LIN {X 0,Y 573.23,Z 214.707,A -85,B 0,C 180,E1 -2343.515,E2 -2343.515} C_VEL
LIN {X 0,Y 573.292,Z 214.696,A -85,B 0,C 180,E1 -2345.628,E2 -2345.628} C_VEL
LIN {X 0,Y 573.285,Z 214.699,A -85,B 0,C 180,E1 -2348.46,E2 -2348.46} C_VEL
LIN {X 0,Y 573.275,Z 214.705,A -85,B 0,C 180,E1 -2351.312,E2 -2351.312} C_VEL
LIN {X 0,Y 573.259,Z 214.704,A -85,B 0,C 180,E1 -2354.414,E2 -2354.414} C_VEL
LIN {X 0,Y 573.261,Z 214.7,A -85,B 0,C 180,E1 -2357.112,E2 -2357.112} C_VEL
LIN {X 0,Y 573.238,Z 214.703,A -85,B 0,C 180,E1 -2360.077,E2 -2360.077} C_VEL
LIN {X 0,Y 573.221,Z 214.707,A -85,B 0,C 180,E1 -2362.339,E2 -2362.339} C_VEL
LIN {X 0,Y 573.248,Z 214.702,A -85,B 0,C 180,E1 -2364.39,E2 -2364.39} C_VEL
LIN {X 0,Y 572.625,Z 214.783,A -85,B 0,C 180,E1 -2364.976,E2 -2364.976} C_VEL
LIN {X 0,Y 569.778,Z 215.141,A -85,B 0,C 180,E1 -2365.927,E2 -2365.927} C_VEL
LIN {X 0,Y 567.338,Z 215.445,A -85,B 0,C 180,E1 -2366.693,E2 -2366.693} C_VEL
LIN {X 0,Y 566.279,Z 215.573,A -85,B 0,C 180,E1 -2367.284,E2 -2367.284} C_VEL
LIN {X 0,Y 566.188,Z 215.583,A -85,B 0,C 180,E1 -2367.484,E2 -2367.484} C_VEL
LIN {X 0,Y 566.196,Z 215.58,A -85,B 0,C 180,E1 -2369.769,E2 -2369.769} C_VEL
LIN {X 0,Y 566.205,Z 215.585,A -85,B 0,C 180,E1 -2372.43,E2 -2372.43} C_VEL
LIN {X 0,Y 566.182,Z 215.582,A -85,B 0,C 180,E1 -2374.989,E2 -2374.989} C_VEL
LIN {X 0,Y 566.198,Z 215.584,A -85,B 0,C 180,E1 -2377.461,E2 -2377.461} C_VEL
LIN {X 0,Y 566.208,Z 215.581,A -85,B 0,C 180,E1 -2380.199,E2 -2380.199} C_VEL
LIN {X 0,Y 566.198,Z 215.58,A -85,B 0,C 180,E1 -2383.055,E2 -2383.055} C_VEL
LIN {X 0,Y 566.196,Z 215.581,A -85,B 0,C 180,E1 -2386.049,E2 -2386.049} C_VEL
LIN {X 0,Y 566.206,Z 215.58,A -85,B 0,C 180,E1 -2389.215,E2 -2389.215} C_VEL
LIN {X 0,Y 566.158,Z 215.588,A -85,B 0,C 180,E1 -2391.449,E2 -2391.449} C_VEL
LIN {X 0,Y 566.211,Z 219.363,A -85,B 0,C 180,E1 -2393.785,E2 -2393.785} C_VEL
LIN {X 0,Y 566.182,Z 223.459,A -85,B 0,C 180,E1 -2396.271,E2 -2396.271} C_VEL
LIN {X 0,Y 566.113,Z 227.943,A -85,B 0,C 180,E1 -2398.937,E2 -2398.937} C_VEL
LIN {X 0,Y 566.059,Z 232.969,A -85,B 0,C 180,E1 -2401.849,E2 -2401.849} C_VEL
LIN {X 0,Y 566.043,Z 238.59,A -85,B 0,C 180,E1 -2405.03,E2 -2405.03} C_VEL
LIN {X 0,Y 565.994,Z 242.827,A -85,B 0,C 180,E1 -2407.361,E2 -2407.361} C_VEL
LIN {X 0,Y 565.932,Z 247.064,A -85,B 0,C 180,E1 -2409.652,E2 -2409.652} C_VEL
LIN {X 0,Y 565.945,Z 251.369,A -85,B 0,C 180,E1 -2411.913,E2 -2411.913} C_VEL
LIN {X 0,Y 565.953,Z 256.885,A -85,B 0,C 180,E1 -2414.769,E2 -2414.769} C_VEL
LIN {X 0,Y 567.409,Z 265.07,A -85,B 0,C 180,E1 -2414.964,E2 -2414.964} C_VEL
LIN {X 0,Y 567.246,Z 279.422,A -85,B 0,C 180,E1 -2415.331,E2 -2415.331} C_VEL
LIN {X 0,Y 567.109,Z 293.099,A -85,B 0,C 180,E1 -2415.833,E2 -2415.833} C_VEL
LIN {X 0,Y 566.885,Z 306.271,A -85,B 0,C 180,E1 -2416.467,E2 -2416.467} C_VEL
LIN {X 0,Y 566.722,Z 318.211,A -85,B 0,C 180,E1 -2417.193,E2 -2417.193} C_VEL
LIN {X 0,Y 566.536,Z 330.289,A -85,B 0,C 180,E1 -2418.098,E2 -2418.098} C_VEL
LIN {X 0,Y 566.4,Z 341.502,A -85,B 0,C 180,E1 -2419.126,E2 -2419.126} C_VEL
LIN {X 0,Y 566.201,Z 350.968,A -85,B 0,C 180,E1 -2420.173,E2 -2420.173} C_VEL
LIN {X 0,Y 566.123,Z 359.1,A -85,B 0,C 180,E1 -2421.253,E2 -2421.253} C_VEL
LIN {X 0,Y 566.016,Z 366.883,A -85,B 0,C 180,E1 -2422.509,E2 -2422.509} C_VEL
LIN {X 0,Y 565.945,Z 372.324,A -85,B 0,C 180,E1 -2423.583,E2 -2423.583} C_VEL
LIN {X 0,Y 565.928,Z 376.8,A -85,B 0,C 180,E1 -2424.656,E2 -2424.656} C_VEL
LIN {X 0,Y 565.956,Z 380.312,A -85,B 0,C 180,E1 -2425.727,E2 -2425.727} C_VEL
LIN {X 0,Y 565.876,Z 383.744,A -85,B 0,C 180,E1 -2427.153,E2 -2427.153} C_VEL
LIN {X 0,Y 565.843,Z 385.785,A -85,B 0,C 180,E1 -2428.577,E2 -2428.577} C_VEL
LIN {X 0,Y 565.837,Z 386.496,A -85,B 0,C 180,E1 -2430,E2 -2430} C_VEL
LIN {X 0,Y 565.841,Z 385.88,A -85,B 0,C 180,E1 -2431.424,E2 -2431.424} C_VEL
LIN {X 0,Y 565.874,Z 383.922,A -85,B 0,C 180,E1 -2432.848,E2 -2432.848} C_VEL
LIN {X 0,Y 565.957,Z 380.576,A -85,B 0,C 180,E1 -2434.273,E2 -2434.273} C_VEL
LIN {X 0,Y 565.983,Z 375.747,A -85,B 0,C 180,E1 -2435.701,E2 -2435.701} C_VEL
LIN {X 0,Y 565.981,Z 369.281,A -85,B 0,C 180,E1 -2437.133,E2 -2437.133} C_VEL
LIN {X 0,Y 566.093,Z 362.081,A -85,B 0,C 180,E1 -2438.388,E2 -2438.388} C_VEL
LIN {X 0,Y 566.172,Z 354.54,A -85,B 0,C 180,E1 -2439.467,E2 -2439.467} C_VEL
LIN {X 0,Y 566.29,Z 345.484,A -85,B 0,C 180,E1 -2440.548,E2 -2440.548} C_VEL
LIN {X 0,Y 566.471,Z 334.519,A -85,B 0,C 180,E1 -2441.631,E2 -2441.631} C_VEL
LIN {X 0,Y 566.644,Z 323.343,A -85,B 0,C 180,E1 -2442.536,E2 -2442.536} C_VEL
LIN {X 0,Y 566.854,Z 310.99,A -85,B 0,C 180,E1 -2443.351,E2 -2443.351} C_VEL
LIN {X 0,Y 566.995,Z 299.106,A -85,B 0,C 180,E1 -2443.987,E2 -2443.987} C_VEL
LIN {X 0,Y 567.178,Z 285.584,A -85,B 0,C 180,E1 -2444.551,E2 -2444.551} C_VEL
LIN {X 0,Y 567.354,Z 272.078,A -85,B 0,C 180,E1 -2444.965,E2 -2444.965} C_VEL
LIN {X 0,Y 567.197,Z 263.074,A -85,B 0,C 180,E1 -2445.172,E2 -2445.172} C_VEL
LIN {X 0,Y 565.917,Z 256.881,A -85,B 0,C 180,E1 -2445.325,E2 -2445.325} C_VEL
LIN {X 0,Y 565.944,Z 251.541,A -85,B 0,C 180,E1 -2448.087,E2 -2448.087} C_VEL
LIN {X 0,Y 565.933,Z 247.234,A -85,B 0,C 180,E1 -2450.348,E2 -2450.348} C_VEL
LIN {X 0,Y 566.046,Z 241.879,A -85,B 0,C 180,E1 -2453.251,E2 -2453.251} C_VEL
LIN {X 0,Y 566.008,Z 237.377,A -85,B 0,C 180,E1 -2455.759,E2 -2455.759} C_VEL
LIN {X 0,Y 566.066,Z 233.084,A -85,B 0,C 180,E1 -2458.176,E2 -2458.176} C_VEL
LIN {X 0,Y 566.12,Z 227.472,A -85,B 0,C 180,E1 -2461.427,E2 -2461.427} C_VEL
LIN {X 0,Y 566.181,Z 223.231,A -85,B 0,C 180,E1 -2463.958,E2 -2463.958} C_VEL
LIN {X 0,Y 566.226,Z 218.933,A -85,B 0,C 180,E1 -2466.568,E2 -2466.568} C_VEL
LIN {X 0,Y 566.148,Z 215.738,A -85,B 0,C 180,E1 -2468.55,E2 -2468.55} C_VEL
LIN {X 0,Y 566.206,Z 215.581,A -85,B 0,C 180,E1 -2470.785,E2 -2470.785} C_VEL
LIN {X 0,Y 566.197,Z 215.58,A -85,B 0,C 180,E1 -2473.951,E2 -2473.951} C_VEL
LIN {X 0,Y 566.204,Z 215.58,A -85,B 0,C 180,E1 -2477.083,E2 -2477.083} C_VEL
LIN {X 0,Y 566.212,Z 215.578,A -85,B 0,C 180,E1 -2480.315,E2 -2480.315} C_VEL
LIN {X 0,Y 566.203,Z 215.579,A -85,B 0,C 180,E1 -2483.43,E2 -2483.43} C_VEL
LIN {X 0,Y 566.201,Z 215.583,A -85,B 0,C 180,E1 -2486.268,E2 -2486.268} C_VEL
LIN {X 0,Y 566.183,Z 215.584,A -85,B 0,C 180,E1 -2488.926,E2 -2488.926} C_VEL
LIN {X 0,Y 566.197,Z 215.58,A -85,B 0,C 180,E1 -2491.856,E2 -2491.856} C_VEL
LIN {X 0,Y 566.217,Z 215.582,A -85,B 0,C 180,E1 -2494.251,E2 -2494.251} C_VEL
LIN {X 0,Y 566.171,Z 215.583,A -85,B 0,C 180,E1 -2496.72,E2 -2496.72} C_VEL
LIN {X 0,Y 566.205,Z 215.579,A -85,B 0,C 180,E1 -2499.662,E2 -2499.662} C_VEL
LIN {X 0,Y 566.201,Z 215.581,A -85,B 0,C 180,E1 -2502.668,E2 -2502.668} C_VEL
LIN {X 0,Y 566.231,Z 215.58,A -85,B 0,C 180,E1 -2505.627,E2 -2505.627} C_VEL
LIN {X 0,Y 566.239,Z 215.581,A -85,B 0,C 180,E1 -2508.676,E2 -2508.676} C_VEL
LIN {X 0,Y 566.208,Z 215.579,A -85,B 0,C 180,E1 -2511.434,E2 -2511.434} C_VEL
LIN {X 0,Y 566.261,Z 215.572,A -85,B 0,C 180,E1 -2514.302,E2 -2514.302} C_VEL
LIN {X 0,Y 566.264,Z 215.572,A -85,B 0,C 180,E1 -2517.866,E2 -2517.866} C_VEL
LIN {X 0,Y 566.303,Z 215.567,A -85,B 0,C 180,E1 -2520.711,E2 -2520.711} C_VEL
LIN {X 0,Y 566.276,Z 215.571,A -85,B 0,C 180,E1 -2522.845,E2 -2522.845} C_VEL
LIN {X 0,Y 566.245,Z 215.574,A -85,B 0,C 180,E1 -2525.698,E2 -2525.698} C_VEL
LIN {X 0,Y 566.195,Z 215.582,A -85,B 0,C 180,E1 -2528.566,E2 -2528.566} C_VEL
LIN {X 0,Y 566.246,Z 215.58,A -85,B 0,C 180,E1 -2531.454,E2 -2531.454} C_VEL
LIN {X 0,Y 566.241,Z 215.579,A -85,B 0,C 180,E1 -2534.507,E2 -2534.507} C_VEL
LIN {X 0,Y 566.174,Z 215.583,A -85,B 0,C 180,E1 -2537.332,E2 -2537.332} C_VEL
LIN {X 0,Y 566.205,Z 215.585,A -85,B 0,C 180,E1 -2539.581,E2 -2539.581} C_VEL
LIN {X 0,Y 566.198,Z 215.58,A -85,B 0,C 180,E1 -2541.862,E2 -2541.862} C_VEL
LIN {X 0,Y 566.222,Z 215.576,A -85,B 0,C 180,E1 -2545.03,E2 -2545.03} C_VEL
LIN {X 0,Y 566.162,Z 215.587,A -85,B 0,C 180,E1 -2547.342,E2 -2547.342} C_VEL
LIN {X 0,Y 566.175,Z 215.583,A -85,B 0,C 180,E1 -2549.77,E2 -2549.77} C_VEL
LIN {X 0,Y 566.212,Z 215.584,A -85,B 0,C 180,E1 -2552.431,E2 -2552.431} C_VEL
LIN {X 0,Y 566.172,Z 215.584,A -85,B 0,C 180,E1 -2554.988,E2 -2554.988} C_VEL
LIN {X 0,Y 566.192,Z 215.586,A -85,B 0,C 180,E1 -2557.461,E2 -2557.461} C_VEL
LIN {X 0,Y 566.209,Z 215.581,A -85,B 0,C 180,E1 -2560.199,E2 -2560.199} C_VEL
LIN {X 0,Y 566.203,Z 215.581,A -85,B 0,C 180,E1 -2563.054,E2 -2563.054} C_VEL
LIN {X 0,Y 566.157,Z 215.586,A -85,B 0,C 180,E1 -2566.053,E2 -2566.053} C_VEL
LIN {X 0,Y 566.168,Z 215.589,A -85,B 0,C 180,E1 -2568.86,E2 -2568.86} C_VEL
LIN {X 0,Y 566.24,Z 215.762,A -85,B 0,C 180,E1 -2570.728,E2 -2570.728} C_VEL
LIN {X 0,Y 566.486,Z 219.701,A -85,B 0,C 180,E1 -2572.561,E2 -2572.561} C_VEL
LIN {X 0,Y 566.391,Z 226.653,A -85,B 0,C 180,E1 -2575.626,E2 -2575.626} C_VEL
LIN {X 0,Y 566.34,Z 233.716,A -85,B 0,C 180,E1 -2578.587,E2 -2578.587} C_VEL
LIN {X 0,Y 566.215,Z 239.77,A -85,B 0,C 180,E1 -2581.048,E2 -2581.048} C_VEL
LIN {X 0,Y 566.161,Z 246.859,A -85,B 0,C 180,E1 -2583.853,E2 -2583.853} C_VEL
LIN {X 0,Y 566.078,Z 253.937,A -85,B 0,C 180,E1 -2586.591,E2 -2586.591} C_VEL
LIN {X 0,Y 566.043,Z 261.995,A -85,B 0,C 180,E1 -2589.656,E2 -2589.656} C_VEL
LIN {X 0,Y 565.975,Z 269.986,A -85,B 0,C 180,E1 -2592.661,E2 -2592.661} C_VEL
LIN {X 0,Y 565.935,Z 275.545,A -85,B 0,C 180,E1 -2594.713,E2 -2594.713} C_VEL
LIN {X 0,Y 567.413,Z 283.017,A -85,B 0,C 180,E1 -2594.877,E2 -2594.877} C_VEL
LIN {X 0,Y 567.263,Z 297.785,A -85,B 0,C 180,E1 -2595.237,E2 -2595.237} C_VEL
LIN {X 0,Y 567.045,Z 311.961,A -85,B 0,C 180,E1 -2595.739,E2 -2595.739} C_VEL
LIN {X 0,Y 566.872,Z 325.392,A -85,B 0,C 180,E1 -2596.375,E2 -2596.375} C_VEL
LIN {X 0,Y 566.721,Z 337.512,A -85,B 0,C 180,E1 -2597.102,E2 -2597.102} C_VEL
LIN {X 0,Y 566.542,Z 349.749,A -85,B 0,C 180,E1 -2598.007,E2 -2598.007} C_VEL
LIN {X 0,Y 566.433,Z 360.501,A -85,B 0,C 180,E1 -2598.98,E2 -2598.98} C_VEL
LIN {X 0,Y 566.206,Z 369.851,A -85,B 0,C 180,E1 -2599.993,E2 -2599.993} C_VEL
LIN {X 0,Y 566.137,Z 378.172,A -85,B 0,C 180,E1 -2601.073,E2 -2601.073} C_VEL
LIN {X 0,Y 566.046,Z 386.127,A -85,B 0,C 180,E1 -2602.33,E2 -2602.33} C_VEL
LIN {X 0,Y 565.944,Z 392.527,A -85,B 0,C 180,E1 -2603.583,E2 -2603.583} C_VEL
LIN {X 0,Y 565.927,Z 396.961,A -85,B 0,C 180,E1 -2604.656,E2 -2604.656} C_VEL
LIN {X 0,Y 565.957,Z 400.443,A -85,B 0,C 180,E1 -2605.727,E2 -2605.727} C_VEL
LIN {X 0,Y 565.874,Z 403.832,A -85,B 0,C 180,E1 -2607.152,E2 -2607.152} C_VEL
LIN {X 0,Y 565.841,Z 405.833,A -85,B 0,C 180,E1 -2608.576,E2 -2608.576} C_VEL
LIN {X 0,Y 565.837,Z 406.5,A -85,B 0,C 180,E1 -2610,E2 -2610} C_VEL
LIN {X 0,Y 565.841,Z 405.834,A -85,B 0,C 180,E1 -2611.423,E2 -2611.423} C_VEL
LIN {X 0,Y 565.874,Z 403.834,A -85,B 0,C 180,E1 -2612.848,E2 -2612.848} C_VEL
LIN {X 0,Y 565.957,Z 400.445,A -85,B 0,C 180,E1 -2614.273,E2 -2614.273} C_VEL
LIN {X 0,Y 565.985,Z 395.568,A -85,B 0,C 180,E1 -2615.701,E2 -2615.701} C_VEL
LIN {X 0,Y 565.995,Z 391.044,A -85,B 0,C 180,E1 -2616.739,E2 -2616.739} C_VEL
LIN {X 0,Y 566.047,Z 384.037,A -85,B 0,C 180,E1 -2618.029,E2 -2618.029} C_VEL
LIN {X 0,Y 566.177,Z 375.558,A -85,B 0,C 180,E1 -2619.286,E2 -2619.286} C_VEL
LIN {X 0,Y 566.294,Z 366.707,A -85,B 0,C 180,E1 -2620.367,E2 -2620.367} C_VEL
LIN {X 0,Y 566.485,Z 355.989,A -85,B 0,C 180,E1 -2621.449,E2 -2621.449} C_VEL
LIN {X 0,Y 566.653,Z 345.14,A -85,B 0,C 180,E1 -2622.354,E2 -2622.354} C_VEL
LIN {X 0,Y 566.74,Z 333.256,A -85,B 0,C 180,E1 -2623.171,E2 -2623.171} C_VEL
LIN {X 0,Y 566.979,Z 320.096,A -85,B 0,C 180,E1 -2623.896,E2 -2623.896} C_VEL
LIN {X 0,Y 567.184,Z 307.303,A -85,B 0,C 180,E1 -2624.445,E2 -2624.445} C_VEL
LIN {X 0,Y 567.327,Z 293.409,A -85,B 0,C 180,E1 -2624.887,E2 -2624.887} C_VEL
LIN {X 0,Y 567.245,Z 282.071,A -85,B 0,C 180,E1 -2625.146,E2 -2625.146} C_VEL
LIN {X 0,Y 565.934,Z 275.48,A -85,B 0,C 180,E1 -2625.301,E2 -2625.301} C_VEL
LIN {X 0,Y 565.986,Z 267.989,A -85,B 0,C 180,E1 -2628.085,E2 -2628.085} C_VEL
LIN {X 0,Y 566.071,Z 259.998,A -85,B 0,C 180,E1 -2631.103,E2 -2631.103} C_VEL
LIN {X 0,Y 566.111,Z 251.897,A -85,B 0,C 180,E1 -2634.185,E2 -2634.185} C_VEL
LIN {X 0,Y 566.21,Z 243.8,A -85,B 0,C 180,E1 -2637.339,E2 -2637.339} C_VEL
LIN {X 0,Y 566.294,Z 235.712,A -85,B 0,C 180,E1 -2640.586,E2 -2640.586} C_VEL
LIN {X 0,Y 566.355,Z 229.675,A -85,B 0,C 180,E1 -2643.093,E2 -2643.093} C_VEL
LIN {X 0,Y 566.391,Z 223.657,A -85,B 0,C 180,E1 -2645.676,E2 -2645.676} C_VEL
LIN {X 0,Y 566.444,Z 217.719,A -85,B 0,C 180,E1 -2648.343,E2 -2648.343} C_VEL
LIN {X 0,Y 566.219,Z 215.582,A -85,B 0,C 180,E1 -2649.377,E2 -2649.377} C_VEL
LIN {X 0,Y 566.173,Z 215.584,A -85,B 0,C 180,E1 -2652.091,E2 -2652.091} C_VEL
LIN {X 0,Y 566.165,Z 215.587,A -85,B 0,C 180,E1 -2655.037,E2 -2655.037} C_VEL
LIN {X 0,Y 566.212,Z 215.584,A -85,B 0,C 180,E1 -2657.913,E2 -2657.913} C_VEL
LIN {X 0,Y 566.214,Z 215.581,A -85,B 0,C 180,E1 -2660.726,E2 -2660.726} C_VEL
LIN {X 0,Y 566.18,Z 215.583,A -85,B 0,C 180,E1 -2663.429,E2 -2663.429} C_VEL
LIN {X 0,Y 566.213,Z 215.581,A -85,B 0,C 180,E1 -2666.266,E2 -2666.266} C_VEL
LIN {X 0,Y 566.196,Z 215.584,A -85,B 0,C 180,E1 -2668.923,E2 -2668.923} C_VEL
LIN {X 0,Y 566.171,Z 215.584,A -85,B 0,C 180,E1 -2671.855,E2 -2671.855} C_VEL
LIN {X 0,Y 566.239,Z 215.575,A -85,B 0,C 180,E1 -2675.039,E2 -2675.039} C_VEL
LIN {X 0,Y 566.196,Z 215.58,A -85,B 0,C 180,E1 -2678.138,E2 -2678.138} C_VEL
LIN {X 0,Y 566.233,Z 215.581,A -85,B 0,C 180,E1 -2680.614,E2 -2680.614} C_VEL
LIN {X 0,Y 566.167,Z 215.585,A -85,B 0,C 180,E1 -2683.411,E2 -2683.411} C_VEL
LIN {X 0,Y 566.24,Z 215.578,A -85,B 0,C 180,E1 -2685.627,E2 -2685.627} C_VEL
LIN {X 0,Y 566.238,Z 215.58,A -85,B 0,C 180,E1 -2688.675,E2 -2688.675} C_VEL
LIN {X 0,Y 566.196,Z 215.581,A -85,B 0,C 180,E1 -2691.434,E2 -2691.434} C_VEL
LIN {X 0,Y 566.243,Z 215.574,A -85,B 0,C 180,E1 -2694.302,E2 -2694.302} C_VEL
LIN {X 0,Y 566.276,Z 215.572,A -85,B 0,C 180,E1 -2697.155,E2 -2697.155} C_VEL
LIN {X 0,Y 566.293,Z 215.575,A -85,B 0,C 180,E1 -2700,E2 -2700} C_VEL
LIN {X 0,Y 566.258,Z 215.574,A -85,B 0,C 180,E1 -2702.846,E2 -2702.846} C_VEL
LIN {X 0,Y 566.259,Z 215.572,A -85,B 0,C 180,E1 -2705.698,E2 -2705.698} C_VEL
LIN {X 0,Y 566.229,Z 215.577,A -85,B 0,C 180,E1 -2708.566,E2 -2708.566} C_VEL
LIN {X 0,Y 566.242,Z 215.579,A -85,B 0,C 180,E1 -2711.454,E2 -2711.454} C_VEL
LIN {X 0,Y 566.215,Z 215.583,A -85,B 0,C 180,E1 -2714.498,E2 -2714.498} C_VEL
LIN {X 0,Y 566.201,Z 215.58,A -85,B 0,C 180,E1 -2717.332,E2 -2717.332} C_VEL
LIN {X 0,Y 566.205,Z 215.579,A -85,B 0,C 180,E1 -2720.338,E2 -2720.338} C_VEL
LIN {X 0,Y 566.168,Z 215.584,A -85,B 0,C 180,E1 -2723.28,E2 -2723.28} C_VEL
LIN {X 0,Y 566.213,Z 215.582,A -85,B 0,C 180,E1 -2725.749,E2 -2725.749} C_VEL
LIN {X 0,Y 566.188,Z 215.583,A -85,B 0,C 180,E1 -2727.484,E2 -2727.484} C_VEL
LIN {X 0,Y 565.508,Z 215.667,A -85,B 0,C 180,E1 -2728.078,E2 -2728.078} C_VEL
LIN {X 0,Y 562.646,Z 216.027,A -85,B 0,C 180,E1 -2729.042,E2 -2729.042} C_VEL
LIN {X 0,Y 560.24,Z 216.324,A -85,B 0,C 180,E1 -2729.818,E2 -2729.818} C_VEL
LIN {X 0,Y 559.214,Z 216.452,A -85,B 0,C 180,E1 -2730.416,E2 -2730.416} C_VEL
LIN {X 0,Y 559.134,Z 216.46,A -85,B 0,C 180,E1 -2730.619,E2 -2730.619} C_VEL
LIN {X 0,Y 559.154,Z 216.46,A -85,B 0,C 180,E1 -2732.716,E2 -2732.716} C_VEL
LIN {X 0,Y 559.13,Z 216.463,A -85,B 0,C 180,E1 -2735.324,E2 -2735.324} C_VEL
LIN {X 0,Y 559.133,Z 216.46,A -85,B 0,C 180,E1 -2738.018,E2 -2738.018} C_VEL
LIN {X 0,Y 559.128,Z 216.464,A -85,B 0,C 180,E1 -2740.815,E2 -2740.815} C_VEL
LIN {X 0,Y 559.139,Z 216.466,A -85,B 0,C 180,E1 -2743.734,E2 -2743.734} C_VEL
LIN {X 0,Y 559.147,Z 216.462,A -85,B 0,C 180,E1 -2746.804,E2 -2746.804} C_VEL
LIN {X 0,Y 559.157,Z 216.458,A -85,B 0,C 180,E1 -2749.188,E2 -2749.188} C_VEL
LIN {X 0,Y 559.124,Z 216.463,A -85,B 0,C 180,E1 -2751.198,E2 -2751.198} C_VEL
LIN {X 0,Y 559.201,Z 218.824,A -85,B 0,C 180,E1 -2752.896,E2 -2752.896} C_VEL
LIN {X 0,Y 559.148,Z 223.949,A -85,B 0,C 180,E1 -2756.054,E2 -2756.054} C_VEL
LIN {X 0,Y 559.064,Z 228.806,A -85,B 0,C 180,E1 -2758.975,E2 -2758.975} C_VEL
LIN {X 0,Y 558.981,Z 233.38,A -85,B 0,C 180,E1 -2761.655,E2 -2761.655} C_VEL
LIN {X 0,Y 558.965,Z 238.679,A -85,B 0,C 180,E1 -2764.692,E2 -2764.692} C_VEL
LIN {X 0,Y 558.944,Z 242.914,A -85,B 0,C 180,E1 -2767.059,E2 -2767.059} C_VEL
LIN {X 0,Y 558.854,Z 247.126,A -85,B 0,C 180,E1 -2769.383,E2 -2769.383} C_VEL
LIN {X 0,Y 558.854,Z 251.37,A -85,B 0,C 180,E1 -2771.676,E2 -2771.676} C_VEL
LIN {X 0,Y 558.852,Z 256.887,A -85,B 0,C 180,E1 -2774.57,E2 -2774.57} C_VEL
LIN {X 0,Y 560.536,Z 265.968,A -85,B 0,C 180,E1 -2774.793,E2 -2774.793} C_VEL
LIN {X 0,Y 560.389,Z 279.941,A -85,B 0,C 180,E1 -2775.163,E2 -2775.163} C_VEL
LIN {X 0,Y 560.209,Z 294.189,A -85,B 0,C 180,E1 -2775.701,E2 -2775.701} C_VEL
LIN {X 0,Y 559.94,Z 307.872,A -85,B 0,C 180,E1 -2776.388,E2 -2776.388} C_VEL
LIN {X 0,Y 559.716,Z 320.802,A -85,B 0,C 180,E1 -2777.214,E2 -2777.214} C_VEL
LIN {X 0,Y 559.523,Z 332.432,A -85,B 0,C 180,E1 -2778.131,E2 -2778.131} C_VEL
LIN {X 0,Y 559.351,Z 342.956,A -85,B 0,C 180,E1 -2779.137,E2 -2779.137} C_VEL
LIN {X 0,Y 559.151,Z 352.457,A -85,B 0,C 180,E1 -2780.231,E2 -2780.231} C_VEL
LIN {X 0,Y 559.029,Z 361.525,A -85,B 0,C 180,E1 -2781.505,E2 -2781.505} C_VEL
LIN {X 0,Y 558.908,Z 368.829,A -85,B 0,C 180,E1 -2782.776,E2 -2782.776} C_VEL
LIN {X 0,Y 558.886,Z 373.939,A -85,B 0,C 180,E1 -2783.864,E2 -2783.864} C_VEL
LIN {X 0,Y 558.821,Z 379.25,A -85,B 0,C 180,E1 -2785.311,E2 -2785.311} C_VEL
LIN {X 0,Y 558.825,Z 382.209,A -85,B 0,C 180,E1 -2786.395,E2 -2786.395} C_VEL
LIN {X 0,Y 558.744,Z 384.935,A -85,B 0,C 180,E1 -2787.838,E2 -2787.838} C_VEL
LIN {X 0,Y 558.737,Z 386.306,A -85,B 0,C 180,E1 -2789.279,E2 -2789.279} C_VEL
LIN {X 0,Y 558.739,Z 386.354,A -85,B 0,C 180,E1 -2790.721,E2 -2790.721} C_VEL
LIN {X 0,Y 558.742,Z 385.07,A -85,B 0,C 180,E1 -2792.163,E2 -2792.163} C_VEL
LIN {X 0,Y 558.825,Z 382.426,A -85,B 0,C 180,E1 -2793.605,E2 -2793.605} C_VEL
LIN {X 0,Y 558.821,Z 379.513,A -85,B 0,C 180,E1 -2794.689,E2 -2794.689} C_VEL
LIN {X 0,Y 558.883,Z 374.321,A -85,B 0,C 180,E1 -2796.136,E2 -2796.136} C_VEL
LIN {X 0,Y 558.907,Z 369.278,A -85,B 0,C 180,E1 -2797.224,E2 -2797.224} C_VEL
LIN {X 0,Y 559.029,Z 362.078,A -85,B 0,C 180,E1 -2798.495,E2 -2798.495} C_VEL
LIN {X 0,Y 559.124,Z 354.537,A -85,B 0,C 180,E1 -2799.587,E2 -2799.587} C_VEL
LIN {X 0,Y 559.288,Z 345.478,A -85,B 0,C 180,E1 -2800.682,E2 -2800.682} C_VEL
LIN {X 0,Y 559.482,Z 334.512,A -85,B 0,C 180,E1 -2801.778,E2 -2801.778} C_VEL
LIN {X 0,Y 559.679,Z 323.336,A -85,B 0,C 180,E1 -2802.695,E2 -2802.695} C_VEL
LIN {X 0,Y 559.921,Z 310.983,A -85,B 0,C 180,E1 -2803.52,E2 -2803.52} C_VEL
LIN {X 0,Y 560.106,Z 299.096,A -85,B 0,C 180,E1 -2804.163,E2 -2804.163} C_VEL
LIN {X 0,Y 560.293,Z 286.039,A -85,B 0,C 180,E1 -2804.717,E2 -2804.717} C_VEL
LIN {X 0,Y 560.489,Z 272.334,A -85,B 0,C 180,E1 -2805.146,E2 -2805.146} C_VEL
LIN {X 0,Y 560.381,Z 264.367,A -85,B 0,C 180,E1 -2805.334,E2 -2805.334} C_VEL
LIN {X 0,Y 558.844,Z 256.88,A -85,B 0,C 180,E1 -2805.524,E2 -2805.524} C_VEL
LIN {X 0,Y 558.854,Z 251.54,A -85,B 0,C 180,E1 -2808.324,E2 -2808.324} C_VEL
LIN {X 0,Y 558.853,Z 247.29,A -85,B 0,C 180,E1 -2810.617,E2 -2810.617} C_VEL
LIN {X 0,Y 558.95,Z 242.295,A -85,B 0,C 180,E1 -2813.383,E2 -2813.383} C_VEL
LIN {X 0,Y 558.931,Z 237.446,A -85,B 0,C 180,E1 -2816.11,E2 -2816.11} C_VEL
LIN {X 0,Y 559.018,Z 233.198,A -85,B 0,C 180,E1 -2818.538,E2 -2818.538} C_VEL
LIN {X 0,Y 559.078,Z 228.558,A -85,B 0,C 180,E1 -2821.261,E2 -2821.261} C_VEL
LIN {X 0,Y 559.134,Z 223.286,A -85,B 0,C 180,E1 -2824.446,E2 -2824.446} C_VEL
LIN {X 0,Y 559.202,Z 218.976,A -85,B 0,C 180,E1 -2827.104,E2 -2827.104} C_VEL
LIN {X 0,Y 559.117,Z 216.466,A -85,B 0,C 180,E1 -2828.801,E2 -2828.801} C_VEL
LIN {X 0,Y 559.163,Z 216.46,A -85,B 0,C 180,E1 -2831.051,E2 -2831.051} C_VEL
LIN {X 0,Y 559.141,Z 216.46,A -85,B 0,C 180,E1 -2833.734,E2 -2833.734} C_VEL
LIN {X 0,Y 559.149,Z 216.46,A -85,B 0,C 180,E1 -2836.804,E2 -2836.804} C_VEL
LIN {X 0,Y 559.178,Z 216.455,A -85,B 0,C 180,E1 -2840.134,E2 -2840.134} C_VEL
LIN {X 0,Y 559.144,Z 216.464,A -85,B 0,C 180,E1 -2842.892,E2 -2842.892} C_VEL
LIN {X 0,Y 559.16,Z 216.463,A -85,B 0,C 180,E1 -2846.052,E2 -2846.052} C_VEL
LIN {X 0,Y 559.148,Z 216.461,A -85,B 0,C 180,E1 -2848.98,E2 -2848.98} C_VEL
LIN {X 0,Y 559.147,Z 216.458,A -85,B 0,C 180,E1 -2851.624,E2 -2851.624} C_VEL
LIN {X 0,Y 559.184,Z 216.457,A -85,B 0,C 180,E1 -2853.903,E2 -2853.903} C_VEL
LIN {X 0,Y 559.141,Z 216.459,A -85,B 0,C 180,E1 -2856.572,E2 -2856.572} C_VEL
LIN {X 0,Y 559.175,Z 216.456,A -85,B 0,C 180,E1 -2859.395,E2 -2859.395} C_VEL
LIN {X 0,Y 559.14,Z 216.46,A -85,B 0,C 180,E1 -2861.685,E2 -2861.685} C_VEL
LIN {X 0,Y 559.167,Z 216.461,A -85,B 0,C 180,E1 -2863.948,E2 -2863.948} C_VEL
LIN {X 0,Y 559.165,Z 216.456,A -85,B 0,C 180,E1 -2866.184,E2 -2866.184} C_VEL
LIN {X 0,Y 559.193,Z 216.454,A -85,B 0,C 180,E1 -2869.133,E2 -2869.133} C_VEL
LIN {X 0,Y 559.199,Z 216.457,A -85,B 0,C 180,E1 -2872.053,E2 -2872.053} C_VEL
LIN {X 0,Y 559.254,Z 216.448,A -85,B 0,C 180,E1 -2874.953,E2 -2874.953} C_VEL
LIN {X 0,Y 559.237,Z 216.447,A -85,B 0,C 180,E1 -2877.839,E2 -2877.839} C_VEL
LIN {X 0,Y 559.273,Z 216.443,A -85,B 0,C 180,E1 -2880.72,E2 -2880.72} C_VEL
LIN {X 0,Y 559.242,Z 216.447,A -85,B 0,C 180,E1 -2882.881,E2 -2882.881} C_VEL
LIN {X 0,Y 559.214,Z 216.45,A -85,B 0,C 180,E1 -2885.77,E2 -2885.77} C_VEL
LIN {X 0,Y 559.162,Z 216.457,A -85,B 0,C 180,E1 -2888.675,E2 -2888.675} C_VEL
LIN {X 0,Y 559.21,Z 216.454,A -85,B 0,C 180,E1 -2891.6,E2 -2891.6} C_VEL
LIN {X 0,Y 559.205,Z 216.457,A -85,B 0,C 180,E1 -2894.595,E2 -2894.595} C_VEL
LIN {X 0,Y 559.124,Z 216.463,A -85,B 0,C 180,E1 -2897.558,E2 -2897.558} C_VEL
LIN {X 0,Y 559.168,Z 216.458,A -85,B 0,C 180,E1 -2899.838,E2 -2899.838} C_VEL
LIN {X 0,Y 559.145,Z 216.459,A -85,B 0,C 180,E1 -2902.153,E2 -2902.153} C_VEL
LIN {X 0,Y 559.164,Z 216.455,A -85,B 0,C 180,E1 -2905.183,E2 -2905.183} C_VEL
LIN {X 0,Y 559.114,Z 216.462,A -85,B 0,C 180,E1 -2908.37,E2 -2908.37} C_VEL
LIN {X 0,Y 559.153,Z 216.459,A -85,B 0,C 180,E1 -2911.274,E2 -2911.274} C_VEL
LIN {X 0,Y 559.167,Z 216.46,A -85,B 0,C 180,E1 -2913.949,E2 -2913.949} C_VEL
LIN {X 0,Y 559.131,Z 216.465,A -85,B 0,C 180,E1 -2917.109,E2 -2917.109} C_VEL
LIN {X 0,Y 559.163,Z 216.457,A -85,B 0,C 180,E1 -2919.941,E2 -2919.941} C_VEL
LIN {X 0,Y 559.163,Z 216.458,A -85,B 0,C 180,E1 -2922.743,E2 -2922.743} C_VEL
LIN {X 0,Y 559.124,Z 216.464,A -85,B 0,C 180,E1 -2925.764,E2 -2925.764} C_VEL
LIN {X 0,Y 559.151,Z 216.46,A -85,B 0,C 180,E1 -2928.228,E2 -2928.228} C_VEL
LIN {X 0,Y 559.178,Z 216.474,A -85,B 0,C 180,E1 -2930.485,E2 -2930.485} C_VEL
LIN {X 0,Y 559.483,Z 220.326,A -85,B 0,C 180,E1 -2932.315,E2 -2932.315} C_VEL
LIN {X 0,Y 559.385,Z 225.731,A -85,B 0,C 180,E1 -2934.751,E2 -2934.751} C_VEL
LIN {X 0,Y 559.323,Z 231.73,A -85,B 0,C 180,E1 -2937.338,E2 -2937.338} C_VEL
LIN {X 0,Y 559.238,Z 238.424,A -85,B 0,C 180,E1 -2940.127,E2 -2940.127} C_VEL
LIN {X 0,Y 559.164,Z 245.971,A -85,B 0,C 180,E1 -2943.174,E2 -2943.174} C_VEL
LIN {X 0,Y 559.028,Z 253.857,A -85,B 0,C 180,E1 -2946.278,E2 -2946.278} C_VEL
LIN {X 0,Y 559.017,Z 260.949,A -85,B 0,C 180,E1 -2949.004,E2 -2949.004} C_VEL
LIN {X 0,Y 558.93,Z 267.989,A -85,B 0,C 180,E1 -2951.678,E2 -2951.678} C_VEL
LIN {X 0,Y 558.881,Z 275.545,A -85,B 0,C 180,E1 -2954.515,E2 -2954.515} C_VEL
LIN {X 0,Y 560.569,Z 284.159,A -85,B 0,C 180,E1 -2954.712,E2 -2954.712} C_VEL
LIN {X 0,Y 560.397,Z 298.443,A -85,B 0,C 180,E1 -2955.072,E2 -2955.072} C_VEL
LIN {X 0,Y 560.155,Z 311.962,A -85,B 0,C 180,E1 -2955.56,E2 -2955.56} C_VEL
LIN {X 0,Y 559.961,Z 325.394,A -85,B 0,C 180,E1 -2956.204,E2 -2956.204} C_VEL
LIN {X 0,Y 559.777,Z 337.514,A -85,B 0,C 180,E1 -2956.939,E2 -2956.939} C_VEL
LIN {X 0,Y 559.564,Z 349.748,A -85,B 0,C 180,E1 -2957.855,E2 -2957.855} C_VEL
LIN {X 0,Y 559.413,Z 360.773,A -85,B 0,C 180,E1 -2958.868,E2 -2958.868} C_VEL
LIN {X 0,Y 559.186,Z 369.851,A -85,B 0,C 180,E1 -2959.866,E2 -2959.866} C_VEL
LIN {X 0,Y 559.073,Z 378.173,A -85,B 0,C 180,E1 -2960.959,E2 -2960.959} C_VEL
LIN {X 0,Y 558.973,Z 386.127,A -85,B 0,C 180,E1 -2962.232,E2 -2962.232} C_VEL
LIN {X 0,Y 558.872,Z 392.527,A -85,B 0,C 180,E1 -2963.501,E2 -2963.501} C_VEL
LIN {X 0,Y 558.858,Z 396.96,A -85,B 0,C 180,E1 -2964.588,E2 -2964.588} C_VEL
LIN {X 0,Y 558.866,Z 400.443,A -85,B 0,C 180,E1 -2965.673,E2 -2965.673} C_VEL
LIN {X 0,Y 558.795,Z 403.832,A -85,B 0,C 180,E1 -2967.116,E2 -2967.116} C_VEL
LIN {X 0,Y 558.741,Z 405.833,A -85,B 0,C 180,E1 -2968.558,E2 -2968.558} C_VEL
LIN {X 0,Y 558.738,Z 406.5,A -85,B 0,C 180,E1 -2970,E2 -2970} C_VEL
LIN {X 0,Y 558.741,Z 405.834,A -85,B 0,C 180,E1 -2971.441,E2 -2971.441} C_VEL
LIN {X 0,Y 558.795,Z 403.835,A -85,B 0,C 180,E1 -2972.884,E2 -2972.884} C_VEL
LIN {X 0,Y 558.866,Z 400.446,A -85,B 0,C 180,E1 -2974.327,E2 -2974.327} C_VEL
LIN {X 0,Y 558.914,Z 395.568,A -85,B 0,C 180,E1 -2975.773,E2 -2975.773} C_VEL
LIN {X 0,Y 558.907,Z 389.054,A -85,B 0,C 180,E1 -2977.224,E2 -2977.224} C_VEL
LIN {X 0,Y 559.028,Z 381.802,A -85,B 0,C 180,E1 -2978.495,E2 -2978.495} C_VEL
LIN {X 0,Y 559.146,Z 372.822,A -85,B 0,C 180,E1 -2979.769,E2 -2979.769} C_VEL
LIN {X 0,Y 559.35,Z 363.392,A -85,B 0,C 180,E1 -2980.863,E2 -2980.863} C_VEL
LIN {X 0,Y 559.514,Z 352.953,A -85,B 0,C 180,E1 -2981.87,E2 -2981.87} C_VEL
LIN {X 0,Y 559.716,Z 341.432,A -85,B 0,C 180,E1 -2982.786,E2 -2982.786} C_VEL
LIN {X 0,Y 559.896,Z 328.641,A -85,B 0,C 180,E1 -2983.613,E2 -2983.613} C_VEL
LIN {X 0,Y 560.1,Z 316.149,A -85,B 0,C 180,E1 -2984.256,E2 -2984.256} C_VEL
LIN {X 0,Y 560.367,Z 301.974,A -85,B 0,C 180,E1 -2984.815,E2 -2984.815} C_VEL
LIN {X 0,Y 560.519,Z 287.826,A -85,B 0,C 180,E1 -2985.214,E2 -2985.214} C_VEL
LIN {X 0,Y 560.383,Z 283.021,A -85,B 0,C 180,E1 -2985.317,E2 -2985.317} C_VEL
LIN {X 0,Y 558.864,Z 275.48,A -85,B 0,C 180,E1 -2985.499,E2 -2985.499} C_VEL
LIN {X 0,Y 558.93,Z 267.989,A -85,B 0,C 180,E1 -2988.322,E2 -2988.322} C_VEL
LIN {X 0,Y 559.017,Z 260.949,A -85,B 0,C 180,E1 -2990.996,E2 -2990.996} C_VEL
LIN {X 0,Y 559.044,Z 252.825,A -85,B 0,C 180,E1 -2994.115,E2 -2994.115} C_VEL
LIN {X 0,Y 559.145,Z 245.746,A -85,B 0,C 180,E1 -2996.904,E2 -2996.904} C_VEL
LIN {X 0,Y 559.237,Z 238.411,A -85,B 0,C 180,E1 -2999.873,E2 -2999.873} C_VEL
LIN {X 0,Y 559.321,Z 231.629,A -85,B 0,C 180,E1 -3002.704,E2 -3002.704} C_VEL
LIN {X 0,Y 559.383,Z 225.602,A -85,B 0,C 180,E1 -3005.306,E2 -3005.306} C_VEL
LIN {X 0,Y 559.443,Z 219.657,A -85,B 0,C 180,E1 -3007.993,E2 -3007.993} C_VEL
LIN {X 0,Y 559.195,Z 216.458,A -85,B 0,C 180,E1 -3009.572,E2 -3009.572} C_VEL
LIN {X 0,Y 559.142,Z 216.464,A -85,B 0,C 180,E1 -3012.745,E2 -3012.745} C_VEL
LIN {X 0,Y 559.149,Z 216.461,A -85,B 0,C 180,E1 -3015.761,E2 -3015.761} C_VEL
LIN {X 0,Y 559.186,Z 216.455,A -85,B 0,C 180,E1 -3018.232,E2 -3018.232} C_VEL
LIN {X 0,Y 559.173,Z 216.46,A -85,B 0,C 180,E1 -3021.192,E2 -3021.192} C_VEL
LIN {X 0,Y 559.118,Z 216.463,A -85,B 0,C 180,E1 -3023.788,E2 -3023.788} C_VEL
LIN {X 0,Y 559.164,Z 216.457,A -85,B 0,C 180,E1 -3026.425,E2 -3026.425} C_VEL
LIN {X 0,Y 559.16,Z 216.461,A -85,B 0,C 180,E1 -3028.981,E2 -3028.981} C_VEL
LIN {X 0,Y 559.118,Z 216.462,A -85,B 0,C 180,E1 -3031.629,E2 -3031.629} C_VEL
LIN {X 0,Y 559.156,Z 216.457,A -85,B 0,C 180,E1 -3034.701,E2 -3034.701} C_VEL
LIN {X 0,Y 559.144,Z 216.459,A -85,B 0,C 180,E1 -3037.847,E2 -3037.847} C_VEL
LIN {X 0,Y 559.195,Z 216.458,A -85,B 0,C 180,E1 -3040.494,E2 -3040.494} C_VEL
LIN {X 0,Y 559.144,Z 216.459,A -85,B 0,C 180,E1 -3043.196,E2 -3043.196} C_VEL
LIN {X 0,Y 559.174,Z 216.454,A -85,B 0,C 180,E1 -3046.184,E2 -3046.184} C_VEL
LIN {X 0,Y 559.197,Z 216.452,A -85,B 0,C 180,E1 -3049.134,E2 -3049.134} C_VEL
LIN {X 0,Y 559.141,Z 216.463,A -85,B 0,C 180,E1 -3052.053,E2 -3052.053} C_VEL
LIN {X 0,Y 559.249,Z 216.45,A -85,B 0,C 180,E1 -3054.953,E2 -3054.953} C_VEL
LIN {X 0,Y 559.253,Z 216.446,A -85,B 0,C 180,E1 -3057.839,E2 -3057.839} C_VEL
LIN {X 0,Y 559.262,Z 216.444,A -85,B 0,C 180,E1 -3060.72,E2 -3060.72} C_VEL
LIN {X 0,Y 559.226,Z 216.45,A -85,B 0,C 180,E1 -3062.882,E2 -3062.882} C_VEL
LIN {X 0,Y 559.229,Z 216.448,A -85,B 0,C 180,E1 -3065.77,E2 -3065.77} C_VEL
LIN {X 0,Y 559.188,Z 216.453,A -85,B 0,C 180,E1 -3068.674,E2 -3068.674} C_VEL
LIN {X 0,Y 559.204,Z 216.454,A -85,B 0,C 180,E1 -3071.601,E2 -3071.601} C_VEL
LIN {X 0,Y 559.183,Z 216.46,A -85,B 0,C 180,E1 -3074.588,E2 -3074.588} C_VEL
LIN {X 0,Y 559.161,Z 216.459,A -85,B 0,C 180,E1 -3077.557,E2 -3077.557} C_VEL
LIN {X 0,Y 559.166,Z 216.457,A -85,B 0,C 180,E1 -3079.838,E2 -3079.838} C_VEL
LIN {X 0,Y 559.135,Z 216.46,A -85,B 0,C 180,E1 -3082.153,E2 -3082.153} C_VEL
LIN {X 0,Y 559.178,Z 216.454,A -85,B 0,C 180,E1 -3085.298,E2 -3085.298} C_VEL
LIN {X 0,Y 559.143,Z 216.463,A -85,B 0,C 180,E1 -3087.714,E2 -3087.714} C_VEL
LIN {X 0,Y 559.134,Z 216.46,A -85,B 0,C 180,E1 -3090.619,E2 -3090.619} C_VEL
LIN {X 0,Y 558.472,Z 216.546,A -85,B 0,C 180,E1 -3091.221,E2 -3091.221} C_VEL
LIN {X 0,Y 555.609,Z 216.902,A -85,B 0,C 180,E1 -3092.197,E2 -3092.197} C_VEL
LIN {X 0,Y 553.197,Z 217.2,A -85,B 0,C 180,E1 -3092.983,E2 -3092.983} C_VEL
LIN {X 0,Y 552.177,Z 217.328,A -85,B 0,C 180,E1 -3093.589,E2 -3093.589} C_VEL
LIN {X 0,Y 552.104,Z 217.338,A -85,B 0,C 180,E1 -3093.795,E2 -3093.795} C_VEL
LIN {X 0,Y 552.107,Z 217.336,A -85,B 0,C 180,E1 -3096.747,E2 -3096.747} C_VEL
LIN {X 0,Y 552.129,Z 217.332,A -85,B 0,C 180,E1 -3099.527,E2 -3099.527} C_VEL
LIN {X 0,Y 552.111,Z 217.338,A -85,B 0,C 180,E1 -3102.428,E2 -3102.428} C_VEL
LIN {X 0,Y 552.096,Z 217.341,A -85,B 0,C 180,E1 -3105.562,E2 -3105.562} C_VEL
LIN {X 0,Y 552.122,Z 217.34,A -85,B 0,C 180,E1 -3108.554,E2 -3108.554} C_VEL
LIN {X 0,Y 552.068,Z 217.41,A -85,B 0,C 180,E1 -3111.407,E2 -3111.407} C_VEL
LIN {X 0,Y 552.164,Z 220.401,A -85,B 0,C 180,E1 -3113.309,E2 -3113.309} C_VEL
LIN {X 0,Y 552.098,Z 224.615,A -85,B 0,C 180,E1 -3115.937,E2 -3115.937} C_VEL
LIN {X 0,Y 552.029,Z 228.88,A -85,B 0,C 180,E1 -3118.539,E2 -3118.539} C_VEL
LIN {X 0,Y 551.921,Z 233.825,A -85,B 0,C 180,E1 -3121.477,E2 -3121.477} C_VEL
LIN {X 0,Y 551.883,Z 238.769,A -85,B 0,C 180,E1 -3124.343,E2 -3124.343} C_VEL
LIN {X 0,Y 551.886,Z 243.001,A -85,B 0,C 180,E1 -3126.748,E2 -3126.748} C_VEL
LIN {X 0,Y 551.795,Z 247.22,A -85,B 0,C 180,E1 -3129.107,E2 -3129.107} C_VEL
LIN {X 0,Y 551.77,Z 251.432,A -85,B 0,C 180,E1 -3131.432,E2 -3131.432} C_VEL
LIN {X 0,Y 551.748,Z 255.677,A -85,B 0,C 180,E1 -3133.726,E2 -3133.726} C_VEL
LIN {X 0,Y 551.752,Z 257.016,A -85,B 0,C 180,E1 -3134.378,E2 -3134.378} C_VEL
LIN {X 0,Y 553.681,Z 266.947,A -85,B 0,C 180,E1 -3134.62,E2 -3134.62} C_VEL
LIN {X 0,Y 553.522,Z 281.089,A -85,B 0,C 180,E1 -3135.011,E2 -3135.011} C_VEL
LIN {X 0,Y 553.31,Z 295.194,A -85,B 0,C 180,E1 -3135.566,E2 -3135.566} C_VEL
LIN {X 0,Y 553.004,Z 307.88,A -85,B 0,C 180,E1 -3136.214,E2 -3136.214} C_VEL
LIN {X 0,Y 552.78,Z 320.808,A -85,B 0,C 180,E1 -3137.051,E2 -3137.051} C_VEL
LIN {X 0,Y 552.546,Z 332.437,A -85,B 0,C 180,E1 -3137.979,E2 -3137.979} C_VEL
LIN {X 0,Y 552.342,Z 342.962,A -85,B 0,C 180,E1 -3138.997,E2 -3138.997} C_VEL
LIN {X 0,Y 552.122,Z 352.462,A -85,B 0,C 180,E1 -3140.105,E2 -3140.105} C_VEL
LIN {X 0,Y 551.964,Z 361.53,A -85,B 0,C 180,E1 -3141.396,E2 -3141.396} C_VEL
LIN {X 0,Y 551.834,Z 368.832,A -85,B 0,C 180,E1 -3142.683,E2 -3142.683} C_VEL
LIN {X 0,Y 551.821,Z 375.393,A -85,B 0,C 180,E1 -3144.152,E2 -3144.152} C_VEL
LIN {X 0,Y 551.76,Z 380.316,A -85,B 0,C 180,E1 -3145.617,E2 -3145.617} C_VEL
LIN {X 0,Y 551.721,Z 383.747,A -85,B 0,C 180,E1 -3147.079,E2 -3147.079} C_VEL
LIN {X 0,Y 551.643,Z 385.787,A -85,B 0,C 180,E1 -3148.54,E2 -3148.54} C_VEL
LIN {X 0,Y 551.639,Z 386.496,A -85,B 0,C 180,E1 -3150,E2 -3150} C_VEL
LIN {X 0,Y 551.64,Z 385.879,A -85,B 0,C 180,E1 -3151.46,E2 -3151.46} C_VEL
LIN {X 0,Y 551.719,Z 383.92,A -85,B 0,C 180,E1 -3152.921,E2 -3152.921} C_VEL
LIN {X 0,Y 551.76,Z 380.574,A -85,B 0,C 180,E1 -3154.383,E2 -3154.383} C_VEL
LIN {X 0,Y 551.819,Z 375.743,A -85,B 0,C 180,E1 -3155.848,E2 -3155.848} C_VEL
LIN {X 0,Y 551.833,Z 369.275,A -85,B 0,C 180,E1 -3157.317,E2 -3157.317} C_VEL
LIN {X 0,Y 551.96,Z 362.075,A -85,B 0,C 180,E1 -3158.604,E2 -3158.604} C_VEL
LIN {X 0,Y 552.067,Z 354.532,A -85,B 0,C 180,E1 -3159.711,E2 -3159.711} C_VEL
LIN {X 0,Y 552.282,Z 345.473,A -85,B 0,C 180,E1 -3160.819,E2 -3160.819} C_VEL
LIN {X 0,Y 552.485,Z 334.505,A -85,B 0,C 180,E1 -3161.93,E2 -3161.93} C_VEL
LIN {X 0,Y 552.73,Z 323.329,A -85,B 0,C 180,E1 -3162.857,E2 -3162.857} C_VEL
LIN {X 0,Y 552.995,Z 310.975,A -85,B 0,C 180,E1 -3163.692,E2 -3163.692} C_VEL
LIN {X 0,Y 553.198,Z 299.086,A -85,B 0,C 180,E1 -3164.344,E2 -3164.344} C_VEL
LIN {X 0,Y 553.414,Z 286.549,A -85,B 0,C 180,E1 -3164.885,E2 -3164.885} C_VEL
LIN {X 0,Y 553.626,Z 272.929,A -85,B 0,C 180,E1 -3165.322,E2 -3165.322} C_VEL
LIN {X 0,Y 553.511,Z 265.192,A -85,B 0,C 180,E1 -3165.512,E2 -3165.512} C_VEL
LIN {X 0,Y 551.74,Z 256.878,A -85,B 0,C 180,E1 -3165.729,E2 -3165.729} C_VEL
LIN {X 0,Y 551.781,Z 253.004,A -85,B 0,C 180,E1 -3167.8,E2 -3167.8} C_VEL
LIN {X 0,Y 551.775,Z 248.785,A -85,B 0,C 180,E1 -3170.115,E2 -3170.115} C_VEL
LIN {X 0,Y 551.842,Z 244.578,A -85,B 0,C 180,E1 -3172.462,E2 -3172.462} C_VEL
LIN {X 0,Y 551.903,Z 239.566,A -85,B 0,C 180,E1 -3175.294,E2 -3175.294} C_VEL
LIN {X 0,Y 551.979,Z 233.951,A -85,B 0,C 180,E1 -3178.534,E2 -3178.534} C_VEL
LIN {X 0,Y 552.03,Z 229.025,A -85,B 0,C 180,E1 -3181.465,E2 -3181.465} C_VEL
LIN {X 0,Y 552.091,Z 224.602,A -85,B 0,C 180,E1 -3184.163,E2 -3184.163} C_VEL
LIN {X 0,Y 552.165,Z 220.466,A -85,B 0,C 180,E1 -3186.743,E2 -3186.743} C_VEL
LIN {X 0,Y 552.079,Z 217.553,A -85,B 0,C 180,E1 -3188.592,E2 -3188.592} C_VEL
LIN {X 0,Y 552.123,Z 217.34,A -85,B 0,C 180,E1 -3191.322,E2 -3191.322} C_VEL
LIN {X 0,Y 552.095,Z 217.339,A -85,B 0,C 180,E1 -3193.482,E2 -3193.482} C_VEL
LIN {X 0,Y 552.11,Z 217.339,A -85,B 0,C 180,E1 -3196.576,E2 -3196.576} C_VEL
LIN {X 0,Y 552.106,Z 217.339,A -85,B 0,C 180,E1 -3199.798,E2 -3199.798} C_VEL
LIN {X 0,Y 552.094,Z 217.338,A -85,B 0,C 180,E1 -3202.336,E2 -3202.336} C_VEL
LIN {X 0,Y 552.086,Z 217.338,A -85,B 0,C 180,E1 -3205.051,E2 -3205.051} C_VEL
LIN {X 0,Y 552.116,Z 217.34,A -85,B 0,C 180,E1 -3207.681,E2 -3207.681} C_VEL
LIN {X 0,Y 552.082,Z 217.338,A -85,B 0,C 180,E1 -3210.233,E2 -3210.233} C_VEL
LIN {X 0,Y 552.141,Z 217.332,A -85,B 0,C 180,E1 -3213,E2 -3213} C_VEL
LIN {X 0,Y 552.116,Z 217.333,A -85,B 0,C 180,E1 -3215.161,E2 -3215.161} C_VEL
LIN {X 0,Y 552.13,Z 217.332,A -85,B 0,C 180,E1 -3218.337,E2 -3218.337} C_VEL
LIN {X 0,Y 552.154,Z 217.335,A -85,B 0,C 180,E1 -3220.674,E2 -3220.674} C_VEL
LIN {X 0,Y 552.117,Z 217.339,A -85,B 0,C 180,E1 -3223.737,E2 -3223.737} C_VEL
LIN {X 0,Y 552.132,Z 217.332,A -85,B 0,C 180,E1 -3226.004,E2 -3226.004} C_VEL
LIN {X 0,Y 552.162,Z 217.331,A -85,B 0,C 180,E1 -3228.993,E2 -3228.993} C_VEL
LIN {X 0,Y 552.154,Z 217.335,A -85,B 0,C 180,E1 -3231.951,E2 -3231.951} C_VEL
LIN {X 0,Y 552.229,Z 217.322,A -85,B 0,C 180,E1 -3234.889,E2 -3234.889} C_VEL
LIN {X 0,Y 552.21,Z 217.322,A -85,B 0,C 180,E1 -3237.812,E2 -3237.812} C_VEL
LIN {X 0,Y 552.244,Z 217.318,A -85,B 0,C 180,E1 -3240.729,E2 -3240.729} C_VEL
LIN {X 0,Y 552.209,Z 217.324,A -85,B 0,C 180,E1 -3242.918,E2 -3242.918} C_VEL
LIN {X 0,Y 552.184,Z 217.325,A -85,B 0,C 180,E1 -3245.844,E2 -3245.844} C_VEL
LIN {X 0,Y 552.135,Z 217.332,A -85,B 0,C 180,E1 -3248.786,E2 -3248.786} C_VEL
LIN {X 0,Y 552.167,Z 217.33,A -85,B 0,C 180,E1 -3251.75,E2 -3251.75} C_VEL
LIN {X 0,Y 552.139,Z 217.336,A -85,B 0,C 180,E1 -3254.748,E2 -3254.748} C_VEL
LIN {X 0,Y 552.085,Z 217.343,A -85,B 0,C 180,E1 -3257.789,E2 -3257.789} C_VEL
LIN {X 0,Y 552.129,Z 217.333,A -85,B 0,C 180,E1 -3260.101,E2 -3260.101} C_VEL
LIN {X 0,Y 552.097,Z 217.339,A -85,B 0,C 180,E1 -3262.451,E2 -3262.451} C_VEL
LIN {X 0,Y 552.124,Z 217.332,A -85,B 0,C 180,E1 -3265.342,E2 -3265.342} C_VEL
LIN {X 0,Y 552.082,Z 217.338,A -85,B 0,C 180,E1 -3268.553,E2 -3268.553} C_VEL
LIN {X 0,Y 552.114,Z 217.334,A -85,B 0,C 180,E1 -3271.475,E2 -3271.475} C_VEL
LIN {X 0,Y 552.132,Z 217.338,A -85,B 0,C 180,E1 -3274.17,E2 -3274.17} C_VEL
LIN {X 0,Y 552.099,Z 217.337,A -85,B 0,C 180,E1 -3276.748,E2 -3276.748} C_VEL
LIN {X 0,Y 552.131,Z 217.333,A -85,B 0,C 180,E1 -3279.527,E2 -3279.527} C_VEL
LIN {X 0,Y 552.134,Z 217.337,A -85,B 0,C 180,E1 -3282.425,E2 -3282.425} C_VEL
LIN {X 0,Y 552.076,Z 217.345,A -85,B 0,C 180,E1 -3285.56,E2 -3285.56} C_VEL
LIN {X 0,Y 552.11,Z 217.34,A -85,B 0,C 180,E1 -3288.553,E2 -3288.553} C_VEL
LIN {X 0,Y 552.171,Z 217.428,A -85,B 0,C 180,E1 -3290.358,E2 -3290.358} C_VEL
LIN {X 0,Y 552.489,Z 221.609,A -85,B 0,C 180,E1 -3292.368,E2 -3292.368} C_VEL
LIN {X 0,Y 552.359,Z 229.2,A -85,B 0,C 180,E1 -3295.795,E2 -3295.795} C_VEL
LIN {X 0,Y 552.265,Z 235.599,A -85,B 0,C 180,E1 -3298.55,E2 -3298.55} C_VEL
LIN {X 0,Y 552.133,Z 242.539,A -85,B 0,C 180,E1 -3301.437,E2 -3301.437} C_VEL
LIN {X 0,Y 552.059,Z 248.736,A -85,B 0,C 180,E1 -3303.947,E2 -3303.947} C_VEL
LIN {X 0,Y 551.978,Z 255.791,A -85,B 0,C 180,E1 -3306.752,E2 -3306.752} C_VEL
LIN {X 0,Y 551.905,Z 262.89,A -85,B 0,C 180,E1 -3309.501,E2 -3309.501} C_VEL
LIN {X 0,Y 551.836,Z 269.979,A -85,B 0,C 180,E1 -3312.202,E2 -3312.202} C_VEL
LIN {X 0,Y 551.777,Z 275.545,A -85,B 0,C 180,E1 -3314.311,E2 -3314.311} C_VEL
LIN {X 0,Y 553.729,Z 285.298,A -85,B 0,C 180,E1 -3314.542,E2 -3314.542} C_VEL
LIN {X 0,Y 553.534,Z 299.124,A -85,B 0,C 180,E1 -3314.904,E2 -3314.904} C_VEL
LIN {X 0,Y 553.255,Z 313.087,A -85,B 0,C 180,E1 -3315.423,E2 -3315.423} C_VEL
LIN {X 0,Y 553.058,Z 325.396,A -85,B 0,C 180,E1 -3316.028,E2 -3316.028} C_VEL
LIN {X 0,Y 552.82,Z 337.515,A -85,B 0,C 180,E1 -3316.771,E2 -3316.771} C_VEL
LIN {X 0,Y 552.599,Z 349.746,A -85,B 0,C 180,E1 -3317.7,E2 -3317.7} C_VEL
LIN {X 0,Y 552.4,Z 361.052,A -85,B 0,C 180,E1 -3318.754,E2 -3318.754} C_VEL
LIN {X 0,Y 552.121,Z 371.337,A -85,B 0,C 180,E1 -3319.92,E2 -3319.92} C_VEL
LIN {X 0,Y 552.011,Z 379.405,A -85,B 0,C 180,E1 -3321.027,E2 -3321.027} C_VEL
LIN {X 0,Y 551.901,Z 387.134,A -85,B 0,C 180,E1 -3322.316,E2 -3322.316} C_VEL
LIN {X 0,Y 551.785,Z 393.634,A -85,B 0,C 180,E1 -3323.669,E2 -3323.669} C_VEL
LIN {X 0,Y 551.715,Z 398.201,A -85,B 0,C 180,E1 -3324.884,E2 -3324.884} C_VEL
LIN {X 0,Y 551.74,Z 402.316,A -85,B 0,C 180,E1 -3326.348,E2 -3326.348} C_VEL
LIN {X 0,Y 551.655,Z 405.002,A -85,B 0,C 180,E1 -3327.81,E2 -3327.81} C_VEL
LIN {X 0,Y 551.636,Z 406.333,A -85,B 0,C 180,E1 -3329.27,E2 -3329.27} C_VEL
LIN {X 0,Y 551.636,Z 406.334,A -85,B 0,C 180,E1 -3330.73,E2 -3330.73} C_VEL
LIN {X 0,Y 551.655,Z 405.004,A -85,B 0,C 180,E1 -3332.19,E2 -3332.19} C_VEL
LIN {X 0,Y 551.74,Z 402.32,A -85,B 0,C 180,E1 -3333.652,E2 -3333.652} C_VEL
LIN {X 0,Y 551.715,Z 398.202,A -85,B 0,C 180,E1 -3335.116,E2 -3335.116} C_VEL
LIN {X 0,Y 551.798,Z 393.574,A -85,B 0,C 180,E1 -3336.344,E2 -3336.344} C_VEL
LIN {X 0,Y 551.901,Z 387.135,A -85,B 0,C 180,E1 -3337.684,E2 -3337.684} C_VEL
LIN {X 0,Y 552.011,Z 379.406,A -85,B 0,C 180,E1 -3338.973,E2 -3338.973} C_VEL
LIN {X 0,Y 552.121,Z 371.338,A -85,B 0,C 180,E1 -3340.08,E2 -3340.08} C_VEL
LIN {X 0,Y 552.401,Z 361.09,A -85,B 0,C 180,E1 -3341.242,E2 -3341.242} C_VEL
LIN {X 0,Y 552.598,Z 349.747,A -85,B 0,C 180,E1 -3342.3,E2 -3342.3} C_VEL
LIN {X 0,Y 552.82,Z 337.52,A -85,B 0,C 180,E1 -3343.228,E2 -3343.228} C_VEL
LIN {X 0,Y 553.057,Z 325.402,A -85,B 0,C 180,E1 -3343.972,E2 -3343.972} C_VEL
LIN {X 0,Y 553.306,Z 311.955,A -85,B 0,C 180,E1 -3344.622,E2 -3344.622} C_VEL
LIN {X 0,Y 553.577,Z 297.447,A -85,B 0,C 180,E1 -3345.146,E2 -3345.146} C_VEL
LIN {X 0,Y 553.552,Z 284.163,A -85,B 0,C 180,E1 -3345.487,E2 -3345.487} C_VEL
LIN {X 0,Y 551.778,Z 275.48,A -85,B 0,C 180,E1 -3345.704,E2 -3345.704} C_VEL
LIN {X 0,Y 551.847,Z 267.955,A -85,B 0,C 180,E1 -3348.565,E2 -3348.565} C_VEL
LIN {X 0,Y 551.927,Z 261.877,A -85,B 0,C 180,E1 -3350.888,E2 -3350.888} C_VEL
LIN {X 0,Y 551.993,Z 253.754,A -85,B 0,C 180,E1 -3354.043,E2 -3354.043} C_VEL
LIN {X 0,Y 552.105,Z 246.372,A -85,B 0,C 180,E1 -3356.993,E2 -3356.993} C_VEL
LIN {X 0,Y 552.202,Z 238.896,A -85,B 0,C 180,E1 -3360.066,E2 -3360.066} C_VEL
LIN {X 0,Y 552.309,Z 232.255,A -85,B 0,C 180,E1 -3362.877,E2 -3362.877} C_VEL
LIN {X 0,Y 552.359,Z 226.32,A -85,B 0,C 180,E1 -3365.481,E2 -3365.481} C_VEL
LIN {X 0,Y 552.457,Z 220.955,A -85,B 0,C 180,E1 -3367.934,E2 -3367.934} C_VEL
LIN {X 0,Y 552.155,Z 217.336,A -85,B 0,C 180,E1 -3369.762,E2 -3369.762} C_VEL
LIN {X 0,Y 552.108,Z 217.338,A -85,B 0,C 180,E1 -3372.428,E2 -3372.428} C_VEL
LIN {X 0,Y 552.093,Z 217.339,A -85,B 0,C 180,E1 -3375.562,E2 -3375.562} C_VEL
LIN {X 0,Y 552.132,Z 217.333,A -85,B 0,C 180,E1 -3378.555,E2 -3378.555} C_VEL
LIN {X 0,Y 552.116,Z 217.337,A -85,B 0,C 180,E1 -3381.411,E2 -3381.411} C_VEL
LIN {X 0,Y 552.072,Z 217.345,A -85,B 0,C 180,E1 -3384.155,E2 -3384.155} C_VEL
LIN {X 0,Y 552.123,Z 217.334,A -85,B 0,C 180,E1 -3386.815,E2 -3386.815} C_VEL
LIN {X 0,Y 552.103,Z 217.339,A -85,B 0,C 180,E1 -3389.391,E2 -3389.391} C_VEL
LIN {X 0,Y 552.064,Z 217.341,A -85,B 0,C 180,E1 -3391.899,E2 -3391.899} C_VEL
LIN {X 0,Y 552.123,Z 217.334,A -85,B 0,C 180,E1 -3394.657,E2 -3394.657} C_VEL
LIN {X 0,Y 552.095,Z 217.34,A -85,B 0,C 180,E1 -3397.549,E2 -3397.549} C_VEL
LIN {X 0,Y 552.147,Z 217.335,A -85,B 0,C 180,E1 -3400.375,E2 -3400.375} C_VEL
LIN {X 0,Y 552.107,Z 217.335,A -85,B 0,C 180,E1 -3402.976,E2 -3402.976} C_VEL
LIN {X 0,Y 552.138,Z 217.331,A -85,B 0,C 180,E1 -3406.005,E2 -3406.005} C_VEL
LIN {X 0,Y 552.165,Z 217.329,A -85,B 0,C 180,E1 -3408.993,E2 -3408.993} C_VEL
LIN {X 0,Y 552.111,Z 217.34,A -85,B 0,C 180,E1 -3411.951,E2 -3411.951} C_VEL
LIN {X 0,Y 552.223,Z 217.324,A -85,B 0,C 180,E1 -3414.889,E2 -3414.889} C_VEL
LIN {X 0,Y 552.225,Z 217.321,A -85,B 0,C 180,E1 -3417.812,E2 -3417.812} C_VEL
LIN {X 0,Y 552.234,Z 217.319,A -85,B 0,C 180,E1 -3420.729,E2 -3420.729} C_VEL
LIN {X 0,Y 552.194,Z 217.327,A -85,B 0,C 180,E1 -3422.918,E2 -3422.918} C_VEL
LIN {X 0,Y 552.199,Z 217.324,A -85,B 0,C 180,E1 -3425.844,E2 -3425.844} C_VEL
LIN {X 0,Y 552.155,Z 217.329,A -85,B 0,C 180,E1 -3428.786,E2 -3428.786} C_VEL
LIN {X 0,Y 552.16,Z 217.33,A -85,B 0,C 180,E1 -3431.751,E2 -3431.751} C_VEL
LIN {X 0,Y 552.132,Z 217.336,A -85,B 0,C 180,E1 -3434.749,E2 -3434.749} C_VEL
LIN {X 0,Y 552.111,Z 217.341,A -85,B 0,C 180,E1 -3437.789,E2 -3437.789} C_VEL
LIN {X 0,Y 552.127,Z 217.332,A -85,B 0,C 180,E1 -3440.101,E2 -3440.101} C_VEL
LIN {X 0,Y 552.088,Z 217.341,A -85,B 0,C 180,E1 -3442.451,E2 -3442.451} C_VEL
LIN {X 0,Y 552.158,Z 217.329,A -85,B 0,C 180,E1 -3445.35,E2 -3445.35} C_VEL
LIN {X 0,Y 552.092,Z 217.338,A -85,B 0,C 180,E1 -3448.099,E2 -3448.099} C_VEL
LIN {X 0,Y 552.098,Z 217.34,A -85,B 0,C 180,E1 -3450.616,E2 -3450.616} C_VEL
LIN {X 0,Y 552.109,Z 217.335,A -85,B 0,C 180,E1 -3453.186,E2 -3453.186} C_VEL
LIN {X 0,Y 552.104,Z 217.338,A -85,B 0,C 180,E1 -3453.795,E2 -3453.795} C_VEL
LIN {X 0,Y 551.47,Z 217.421,A -85,B 0,C 180,E1 -3454.403,E2 -3454.403} C_VEL
LIN {X 0,Y 548.651,Z 217.77,A -85,B 0,C 180,E1 -3455.391,E2 -3455.391} C_VEL
LIN {X 0,Y 546.232,Z 218.068,A -85,B 0,C 180,E1 -3456.187,E2 -3456.187} C_VEL
LIN {X 0,Y 545.164,Z 218.201,A -85,B 0,C 180,E1 -3456.8,E2 -3456.8} C_VEL
LIN {X 0,Y 545.063,Z 218.215,A -85,B 0,C 180,E1 -3457.008,E2 -3457.008} C_VEL
LIN {X 0,Y 545.06,Z 218.214,A -85,B 0,C 180,E1 -3460.143,E2 -3460.143} C_VEL
LIN {X 0,Y 545.047,Z 218.215,A -85,B 0,C 180,E1 -3463.11,E2 -3463.11} C_VEL
LIN {X 0,Y 545.051,Z 218.215,A -85,B 0,C 180,E1 -3466.226,E2 -3466.226} C_VEL
LIN {X 0,Y 545.083,Z 218.214,A -85,B 0,C 180,E1 -3468.885,E2 -3468.885} C_VEL
LIN {X 0,Y 545.048,Z 218.218,A -85,B 0,C 180,E1 -3470.815,E2 -3470.815} C_VEL
LIN {X 0,Y 545.066,Z 219.057,A -85,B 0,C 180,E1 -3471.862,E2 -3471.862} C_VEL
LIN {X 0,Y 545.053,Z 222.908,A -85,B 0,C 180,E1 -3474.325,E2 -3474.325} C_VEL
LIN {X 0,Y 545.003,Z 227.104,A -85,B 0,C 180,E1 -3476.951,E2 -3476.951} C_VEL
LIN {X 0,Y 544.918,Z 231.774,A -85,B 0,C 180,E1 -3479.801,E2 -3479.801} C_VEL
LIN {X 0,Y 544.842,Z 236.953,A -85,B 0,C 180,E1 -3482.879,E2 -3482.879} C_VEL
LIN {X 0,Y 544.807,Z 241.678,A -85,B 0,C 180,E1 -3485.619,E2 -3485.619} C_VEL
LIN {X 0,Y 544.761,Z 246.32,A -85,B 0,C 180,E1 -3488.261,E2 -3488.261} C_VEL
LIN {X 0,Y 544.703,Z 251.525,A -85,B 0,C 180,E1 -3491.182,E2 -3491.182} C_VEL
LIN {X 0,Y 544.675,Z 255.748,A -85,B 0,C 180,E1 -3493.509,E2 -3493.509} C_VEL
LIN {X 0,Y 544.672,Z 257.128,A -85,B 0,C 180,E1 -3494.17,E2 -3494.17} C_VEL
LIN {X 0,Y 546.838,Z 267.591,A -85,B 0,C 180,E1 -3494.435,E2 -3494.435} C_VEL
LIN {X 0,Y 546.64,Z 281.971,A -85,B 0,C 180,E1 -3494.849,E2 -3494.849} C_VEL
LIN {X 0,Y 546.418,Z 295.204,A -85,B 0,C 180,E1 -3495.38,E2 -3495.38} C_VEL
LIN {X 0,Y 546.11,Z 307.888,A -85,B 0,C 180,E1 -3496.037,E2 -3496.037} C_VEL
LIN {X 0,Y 545.816,Z 320.814,A -85,B 0,C 180,E1 -3496.883,E2 -3496.883} C_VEL
LIN {X 0,Y 545.552,Z 332.442,A -85,B 0,C 180,E1 -3497.822,E2 -3497.822} C_VEL
LIN {X 0,Y 545.339,Z 342.967,A -85,B 0,C 180,E1 -3498.854,E2 -3498.854} C_VEL
LIN {X 0,Y 545.09,Z 352.466,A -85,B 0,C 180,E1 -3499.976,E2 -3499.976} C_VEL
LIN {X 0,Y 544.911,Z 361.534,A -85,B 0,C 180,E1 -3501.284,E2 -3501.284} C_VEL
LIN {X 0,Y 544.784,Z 368.836,A -85,B 0,C 180,E1 -3502.588,E2 -3502.588} C_VEL
LIN {X 0,Y 544.732,Z 375.395,A -85,B 0,C 180,E1 -3504.076,E2 -3504.076} C_VEL
LIN {X 0,Y 544.655,Z 380.318,A -85,B 0,C 180,E1 -3505.56,E2 -3505.56} C_VEL
LIN {X 0,Y 544.647,Z 383.749,A -85,B 0,C 180,E1 -3507.041,E2 -3507.041} C_VEL
LIN {X 0,Y 544.544,Z 385.788,A -85,B 0,C 180,E1 -3508.521,E2 -3508.521} C_VEL
LIN {X 0,Y 544.54,Z 386.496,A -85,B 0,C 180,E1 -3510,E2 -3510} C_VEL
LIN {X 0,Y 544.541,Z 385.878,A -85,B 0,C 180,E1 -3511.479,E2 -3511.479} C_VEL
LIN {X 0,Y 544.646,Z 383.919,A -85,B 0,C 180,E1 -3512.959,E2 -3512.959} C_VEL
LIN {X 0,Y 544.655,Z 380.572,A -85,B 0,C 180,E1 -3514.44,E2 -3514.44} C_VEL
LIN {X 0,Y 544.729,Z 375.741,A -85,B 0,C 180,E1 -3515.924,E2 -3515.924} C_VEL
LIN {X 0,Y 544.784,Z 369.272,A -85,B 0,C 180,E1 -3517.412,E2 -3517.412} C_VEL
LIN {X 0,Y 544.906,Z 362.071,A -85,B 0,C 180,E1 -3518.717,E2 -3518.717} C_VEL
LIN {X 0,Y 545.04,Z 354.527,A -85,B 0,C 180,E1 -3519.837,E2 -3519.837} C_VEL
LIN {X 0,Y 545.276,Z 345.467,A -85,B 0,C 180,E1 -3520.959,E2 -3520.959} C_VEL
LIN {X 0,Y 545.505,Z 334.498,A -85,B 0,C 180,E1 -3522.085,E2 -3522.085} C_VEL
LIN {X 0,Y 545.787,Z 323.322,A -85,B 0,C 180,E1 -3523.023,E2 -3523.023} C_VEL
LIN {X 0,Y 546.052,Z 310.963,A -85,B 0,C 180,E1 -3523.87,E2 -3523.87} C_VEL
LIN {X 0,Y 546.323,Z 299.073,A -85,B 0,C 180,E1 -3524.528,E2 -3524.528} C_VEL
LIN {X 0,Y 546.544,Z 287.062,A -85,B 0,C 180,E1 -3525.057,E2 -3525.057} C_VEL
LIN {X 0,Y 546.77,Z 273.259,A -85,B 0,C 180,E1 -3525.51,E2 -3525.51} C_VEL
LIN {X 0,Y 546.688,Z 266.472,A -85,B 0,C 180,E1 -3525.683,E2 -3525.683} C_VEL
LIN {X 0,Y 544.678,Z 256.926,A -85,B 0,C 180,E1 -3525.938,E2 -3525.938} C_VEL
LIN {X 0,Y 544.693,Z 253.094,A -85,B 0,C 180,E1 -3528.039,E2 -3528.039} C_VEL
LIN {X 0,Y 544.71,Z 248.877,A -85,B 0,C 180,E1 -3530.387,E2 -3530.387} C_VEL
LIN {X 0,Y 544.796,Z 244.671,A -85,B 0,C 180,E1 -3532.769,E2 -3532.769} C_VEL
LIN {X 0,Y 544.833,Z 239.974,A -85,B 0,C 180,E1 -3535.45,E2 -3535.45} C_VEL
LIN {X 0,Y 544.916,Z 234.398,A -85,B 0,C 180,E1 -3538.714,E2 -3538.714} C_VEL
LIN {X 0,Y 544.963,Z 229.089,A -85,B 0,C 180,E1 -3541.921,E2 -3541.921} C_VEL
LIN {X 0,Y 545.051,Z 224.818,A -85,B 0,C 180,E1 -3544.566,E2 -3544.566} C_VEL
LIN {X 0,Y 545.118,Z 220.505,A -85,B 0,C 180,E1 -3547.298,E2 -3547.298} C_VEL
LIN {X 0,Y 545.053,Z 219.049,A -85,B 0,C 180,E1 -3548.238,E2 -3548.238} C_VEL
LIN {X 0,Y 545.038,Z 218.22,A -85,B 0,C 180,E1 -3549.315,E2 -3549.315} C_VEL
LIN {X 0,Y 545.08,Z 218.211,A -85,B 0,C 180,E1 -3552.103,E2 -3552.103} C_VEL
LIN {X 0,Y 545.039,Z 218.217,A -85,B 0,C 180,E1 -3555.17,E2 -3555.17} C_VEL
LIN {X 0,Y 545.056,Z 218.22,A -85,B 0,C 180,E1 -3557.895,E2 -3557.895} C_VEL
LIN {X 0,Y 545.079,Z 218.213,A -85,B 0,C 180,E1 -3560.818,E2 -3560.818} C_VEL
LIN {X 0,Y 545.045,Z 218.215,A -85,B 0,C 180,E1 -3563.62,E2 -3563.62} C_VEL
LIN {X 0,Y 545.053,Z 218.216,A -85,B 0,C 180,E1 -3566.327,E2 -3566.327} C_VEL
LIN {X 0,Y 545.063,Z 218.215,A -85,B 0,C 180,E1 -3568.952,E2 -3568.952} C_VEL
LIN {X 0,Y 545.084,Z 218.21,A -85,B 0,C 180,E1 -3571.507,E2 -3571.507} C_VEL
LIN {X 0,Y 545.099,Z 218.209,A -85,B 0,C 180,E1 -3574.491,E2 -3574.491} C_VEL
LIN {X 0,Y 545.036,Z 218.221,A -85,B 0,C 180,E1 -3577.242,E2 -3577.242} C_VEL
LIN {X 0,Y 545.119,Z 218.209,A -85,B 0,C 180,E1 -3580.415,E2 -3580.415} C_VEL
LIN {X 0,Y 545.068,Z 218.214,A -85,B 0,C 180,E1 -3583.521,E2 -3583.521} C_VEL
LIN {X 0,Y 545.094,Z 218.211,A -85,B 0,C 180,E1 -3585.82,E2 -3585.82} C_VEL
LIN {X 0,Y 545.119,Z 218.21,A -85,B 0,C 180,E1 -3588.849,E2 -3588.849} C_VEL
LIN {X 0,Y 545.101,Z 218.213,A -85,B 0,C 180,E1 -3591.847,E2 -3591.847} C_VEL
LIN {X 0,Y 545.205,Z 218.196,A -85,B 0,C 180,E1 -3594.823,E2 -3594.823} C_VEL
LIN {X 0,Y 545.184,Z 218.197,A -85,B 0,C 180,E1 -3597.784,E2 -3597.784} C_VEL
LIN {X 0,Y 545.214,Z 218.194,A -85,B 0,C 180,E1 -3600.739,E2 -3600.739} C_VEL
LIN {X 0,Y 545.175,Z 218.2,A -85,B 0,C 180,E1 -3602.956,E2 -3602.956} C_VEL
LIN {X 0,Y 545.134,Z 218.204,A -85,B 0,C 180,E1 -3605.92,E2 -3605.92} C_VEL
LIN {X 0,Y 545.097,Z 218.208,A -85,B 0,C 180,E1 -3608.9,E2 -3608.9} C_VEL
LIN {X 0,Y 545.139,Z 218.204,A -85,B 0,C 180,E1 -3611.904,E2 -3611.904} C_VEL
LIN {X 0,Y 545.087,Z 218.212,A -85,B 0,C 180,E1 -3614.944,E2 -3614.944} C_VEL
LIN {X 0,Y 545.054,Z 218.218,A -85,B 0,C 180,E1 -3618.027,E2 -3618.027} C_VEL
LIN {X 0,Y 545.095,Z 218.209,A -85,B 0,C 180,E1 -3620.372,E2 -3620.372} C_VEL
LIN {X 0,Y 545.085,Z 218.21,A -85,B 0,C 180,E1 -3623.559,E2 -3623.559} C_VEL
LIN {X 0,Y 545.057,Z 218.218,A -85,B 0,C 180,E1 -3626.002,E2 -3626.002} C_VEL
LIN {X 0,Y 545.048,Z 218.215,A -85,B 0,C 180,E1 -3628.739,E2 -3628.739} C_VEL
LIN {X 0,Y 545.063,Z 218.212,A -85,B 0,C 180,E1 -3631.679,E2 -3631.679} C_VEL
LIN {X 0,Y 545.075,Z 218.214,A -85,B 0,C 180,E1 -3634.392,E2 -3634.392} C_VEL
LIN {X 0,Y 545.032,Z 218.223,A -85,B 0,C 180,E1 -3637.304,E2 -3637.304} C_VEL
LIN {X 0,Y 545.068,Z 218.214,A -85,B 0,C 180,E1 -3640.142,E2 -3640.142} C_VEL
LIN {X 0,Y 545.081,Z 218.212,A -85,B 0,C 180,E1 -3643.106,E2 -3643.106} C_VEL
LIN {X 0,Y 545.029,Z 218.218,A -85,B 0,C 180,E1 -3646.229,E2 -3646.229} C_VEL
LIN {X 0,Y 545.072,Z 218.217,A -85,B 0,C 180,E1 -3648.884,E2 -3648.884} C_VEL
LIN {X 0,Y 545.143,Z 218.302,A -85,B 0,C 180,E1 -3650.186,E2 -3650.186} C_VEL
LIN {X 0,Y 545.441,Z 221.612,A -85,B 0,C 180,E1 -3651.812,E2 -3651.812} C_VEL
LIN {X 0,Y 545.342,Z 227.516,A -85,B 0,C 180,E1 -3654.554,E2 -3654.554} C_VEL
LIN {X 0,Y 545.267,Z 233.523,A -85,B 0,C 180,E1 -3657.225,E2 -3657.225} C_VEL
LIN {X 0,Y 545.158,Z 240.574,A -85,B 0,C 180,E1 -3660.242,E2 -3660.242} C_VEL
LIN {X 0,Y 545.081,Z 247.645,A -85,B 0,C 180,E1 -3663.174,E2 -3663.174} C_VEL
LIN {X 0,Y 544.906,Z 255.405,A -85,B 0,C 180,E1 -3666.31,E2 -3666.31} C_VEL
LIN {X 0,Y 544.872,Z 262.804,A -85,B 0,C 180,E1 -3669.224,E2 -3669.224} C_VEL
LIN {X 0,Y 544.766,Z 269.894,A -85,B 0,C 180,E1 -3671.963,E2 -3671.963} C_VEL
LIN {X 0,Y 544.733,Z 275.501,A -85,B 0,C 180,E1 -3674.103,E2 -3674.103} C_VEL
LIN {X 0,Y 546.866,Z 286.887,A -85,B 0,C 180,E1 -3674.376,E2 -3674.376} C_VEL
LIN {X 0,Y 546.719,Z 300.498,A -85,B 0,C 180,E1 -3674.754,E2 -3674.754} C_VEL
LIN {X 0,Y 546.363,Z 314.16,A -85,B 0,C 180,E1 -3675.283,E2 -3675.283} C_VEL
LIN {X 0,Y 546.121,Z 327.051,A -85,B 0,C 180,E1 -3675.942,E2 -3675.942} C_VEL
LIN {X 0,Y 545.864,Z 338.842,A -85,B 0,C 180,E1 -3676.695,E2 -3676.695} C_VEL
LIN {X 0,Y 545.59,Z 350.814,A -85,B 0,C 180,E1 -3677.634,E2 -3677.634} C_VEL
LIN {X 0,Y 545.389,Z 361.67,A -85,B 0,C 180,E1 -3678.673,E2 -3678.673} C_VEL
LIN {X 0,Y 545.101,Z 371.336,A -85,B 0,C 180,E1 -3679.789,E2 -3679.789} C_VEL
LIN {X 0,Y 544.969,Z 379.404,A -85,B 0,C 180,E1 -3680.91,E2 -3680.91} C_VEL
LIN {X 0,Y 544.824,Z 387.133,A -85,B 0,C 180,E1 -3682.216,E2 -3682.216} C_VEL
LIN {X 0,Y 544.753,Z 392.875,A -85,B 0,C 180,E1 -3683.412,E2 -3683.412} C_VEL
LIN {X 0,Y 544.645,Z 398.2,A -85,B 0,C 180,E1 -3684.818,E2 -3684.818} C_VEL
LIN {X 0,Y 544.657,Z 402.316,A -85,B 0,C 180,E1 -3686.301,E2 -3686.301} C_VEL
LIN {X 0,Y 544.57,Z 405.002,A -85,B 0,C 180,E1 -3687.781,E2 -3687.781} C_VEL
LIN {X 0,Y 544.536,Z 406.333,A -85,B 0,C 180,E1 -3689.26,E2 -3689.26} C_VEL
LIN {X 0,Y 544.536,Z 406.334,A -85,B 0,C 180,E1 -3690.739,E2 -3690.739} C_VEL
LIN {X 0,Y 544.57,Z 405.004,A -85,B 0,C 180,E1 -3692.219,E2 -3692.219} C_VEL
LIN {X 0,Y 544.657,Z 402.32,A -85,B 0,C 180,E1 -3693.699,E2 -3693.699} C_VEL
LIN {X 0,Y 544.645,Z 398.202,A -85,B 0,C 180,E1 -3695.182,E2 -3695.182} C_VEL
LIN {X 0,Y 544.738,Z 392.936,A -85,B 0,C 180,E1 -3696.573,E2 -3696.573} C_VEL
LIN {X 0,Y 544.834,Z 386.127,A -85,B 0,C 180,E1 -3697.971,E2 -3697.971} C_VEL
LIN {X 0,Y 544.999,Z 378.175,A -85,B 0,C 180,E1 -3699.276,E2 -3699.276} C_VEL
LIN {X 0,Y 545.175,Z 369.852,A -85,B 0,C 180,E1 -3700.398,E2 -3700.398} C_VEL
LIN {X 0,Y 545.364,Z 360.028,A -85,B 0,C 180,E1 -3701.501,E2 -3701.501} C_VEL
LIN {X 0,Y 545.677,Z 348.648,A -85,B 0,C 180,E1 -3702.553,E2 -3702.553} C_VEL
LIN {X 0,Y 545.886,Z 336.1,A -85,B 0,C 180,E1 -3703.494,E2 -3703.494} C_VEL
LIN {X 0,Y 546.168,Z 323.638,A -85,B 0,C 180,E1 -3704.247,E2 -3704.247} C_VEL
LIN {X 0,Y 546.469,Z 310.823,A -85,B 0,C 180,E1 -3704.857,E2 -3704.857} C_VEL
LIN {X 0,Y 546.723,Z 296.215,A -85,B 0,C 180,E1 -3705.379,E2 -3705.379} C_VEL
LIN {X 0,Y 546.726,Z 285.299,A -85,B 0,C 180,E1 -3705.661,E2 -3705.661} C_VEL
LIN {X 0,Y 544.719,Z 275.455,A -85,B 0,C 180,E1 -3705.912,E2 -3705.912} C_VEL
LIN {X 0,Y 544.781,Z 267.87,A -85,B 0,C 180,E1 -3708.815,E2 -3708.815} C_VEL
LIN {X 0,Y 544.891,Z 260.249,A -85,B 0,C 180,E1 -3711.774,E2 -3711.774} C_VEL
LIN {X 0,Y 544.957,Z 252.653,A -85,B 0,C 180,E1 -3714.78,E2 -3714.78} C_VEL
LIN {X 0,Y 545.102,Z 245.612,A -85,B 0,C 180,E1 -3717.655,E2 -3717.655} C_VEL
LIN {X 0,Y 545.175,Z 239.375,A -85,B 0,C 180,E1 -3720.264,E2 -3720.264} C_VEL
LIN {X 0,Y 545.293,Z 232.785,A -85,B 0,C 180,E1 -3723.096,E2 -3723.096} C_VEL
LIN {X 0,Y 545.347,Z 226.909,A -85,B 0,C 180,E1 -3725.719,E2 -3725.719} C_VEL
LIN {X 0,Y 545.437,Z 221.564,A -85,B 0,C 180,E1 -3728.206,E2 -3728.206} C_VEL
LIN {X 0,Y 545.092,Z 218.214,A -85,B 0,C 180,E1 -3729.925,E2 -3729.925} C_VEL
LIN {X 0,Y 545.038,Z 218.221,A -85,B 0,C 180,E1 -3732.694,E2 -3732.694} C_VEL
LIN {X 0,Y 545.03,Z 218.219,A -85,B 0,C 180,E1 -3735.171,E2 -3735.171} C_VEL
LIN {X 0,Y 545.082,Z 218.216,A -85,B 0,C 180,E1 -3737.897,E2 -3737.897} C_VEL
LIN {X 0,Y 545.08,Z 218.214,A -85,B 0,C 180,E1 -3740.818,E2 -3740.818} C_VEL
LIN {X 0,Y 545.033,Z 218.217,A -85,B 0,C 180,E1 -3743.619,E2 -3743.619} C_VEL
LIN {X 0,Y 545.068,Z 218.214,A -85,B 0,C 180,E1 -3746.328,E2 -3746.328} C_VEL
LIN {X 0,Y 545.068,Z 218.216,A -85,B 0,C 180,E1 -3748.952,E2 -3748.952} C_VEL
LIN {X 0,Y 545.045,Z 218.215,A -85,B 0,C 180,E1 -3751.504,E2 -3751.504} C_VEL
LIN {X 0,Y 545.072,Z 218.213,A -85,B 0,C 180,E1 -3754.497,E2 -3754.497} C_VEL
LIN {X 0,Y 545.04,Z 218.222,A -85,B 0,C 180,E1 -3757.242,E2 -3757.242} C_VEL
LIN {X 0,Y 545.118,Z 218.211,A -85,B 0,C 180,E1 -3760.415,E2 -3760.415} C_VEL
LIN {X 0,Y 545.039,Z 218.218,A -85,B 0,C 180,E1 -3763.52,E2 -3763.52} C_VEL
LIN {X 0,Y 545.098,Z 218.209,A -85,B 0,C 180,E1 -3765.82,E2 -3765.82} C_VEL
LIN {X 0,Y 545.12,Z 218.208,A -85,B 0,C 180,E1 -3768.849,E2 -3768.849} C_VEL
LIN {X 0,Y 545.069,Z 218.218,A -85,B 0,C 180,E1 -3771.846,E2 -3771.846} C_VEL
LIN {X 0,Y 545.199,Z 218.198,A -85,B 0,C 180,E1 -3774.823,E2 -3774.823} C_VEL
LIN {X 0,Y 545.197,Z 218.196,A -85,B 0,C 180,E1 -3777.784,E2 -3777.784} C_VEL
LIN {X 0,Y 545.205,Z 218.195,A -85,B 0,C 180,E1 -3780.739,E2 -3780.739} C_VEL
LIN {X 0,Y 545.162,Z 218.203,A -85,B 0,C 180,E1 -3782.956,E2 -3782.956} C_VEL
LIN {X 0,Y 545.171,Z 218.2,A -85,B 0,C 180,E1 -3785.92,E2 -3785.92} C_VEL
LIN {X 0,Y 545.113,Z 218.206,A -85,B 0,C 180,E1 -3788.9,E2 -3788.9} C_VEL
LIN {X 0,Y 545.103,Z 218.208,A -85,B 0,C 180,E1 -3791.905,E2 -3791.905} C_VEL
LIN {X 0,Y 545.085,Z 218.212,A -85,B 0,C 180,E1 -3794.944,E2 -3794.944} C_VEL
LIN {X 0,Y 545.079,Z 218.214,A -85,B 0,C 180,E1 -3798.026,E2 -3798.026} C_VEL
LIN {X 0,Y 545.093,Z 218.209,A -85,B 0,C 180,E1 -3800.372,E2 -3800.372} C_VEL
LIN {X 0,Y 545.078,Z 218.21,A -85,B 0,C 180,E1 -3803.56,E2 -3803.56} C_VEL
LIN {X 0,Y 545.08,Z 218.216,A -85,B 0,C 180,E1 -3806.001,E2 -3806.001} C_VEL
LIN {X 0,Y 545.076,Z 218.212,A -85,B 0,C 180,E1 -3808.745,E2 -3808.745} C_VEL
LIN {X 0,Y 545.06,Z 218.213,A -85,B 0,C 180,E1 -3811.679,E2 -3811.679} C_VEL
LIN {X 0,Y 545.062,Z 218.214,A -85,B 0,C 180,E1 -3814.565,E2 -3814.565} C_VEL
LIN {X 0,Y 545.063,Z 218.215,A -85,B 0,C 180,E1 -3817.008,E2 -3817.008} C_VEL
LIN {X 0,Y 544.356,Z 218.307,A -85,B 0,C 180,E1 -3817.625,E2 -3817.625} C_VEL
LIN {X 0,Y 541.488,Z 218.662,A -85,B 0,C 180,E1 -3818.626,E2 -3818.626} C_VEL
LIN {X 0,Y 539.092,Z 218.957,A -85,B 0,C 180,E1 -3819.431,E2 -3819.431} C_VEL
LIN {X 0,Y 538.069,Z 219.085,A -85,B 0,C 180,E1 -3820.053,E2 -3820.053} C_VEL
LIN {X 0,Y 537.988,Z 219.094,A -85,B 0,C 180,E1 -3820.264,E2 -3820.264} C_VEL
LIN {X 0,Y 538,Z 219.093,A -85,B 0,C 180,E1 -3822.984,E2 -3822.984} C_VEL
LIN {X 0,Y 538.021,Z 219.091,A -85,B 0,C 180,E1 -3825.927,E2 -3825.927} C_VEL
LIN {X 0,Y 538.032,Z 219.091,A -85,B 0,C 180,E1 -3828.227,E2 -3828.227} C_VEL
LIN {X 0,Y 537.996,Z 219.099,A -85,B 0,C 180,E1 -3830.42,E2 -3830.42} C_VEL
LIN {X 0,Y 537.962,Z 219.1,A -85,B 0,C 180,E1 -3831.165,E2 -3831.165} C_VEL
LIN {X 0,Y 538.076,Z 221.848,A -85,B 0,C 180,E1 -3833.071,E2 -3833.071} C_VEL
LIN {X 0,Y 537.989,Z 226.15,A -85,B 0,C 180,E1 -3835.824,E2 -3835.824} C_VEL
LIN {X 0,Y 537.903,Z 230.425,A -85,B 0,C 180,E1 -3838.492,E2 -3838.492} C_VEL
LIN {X 0,Y 537.809,Z 234.718,A -85,B 0,C 180,E1 -3841.11,E2 -3841.11} C_VEL
LIN {X 0,Y 537.736,Z 238.926,A -85,B 0,C 180,E1 -3843.617,E2 -3843.617} C_VEL
LIN {X 0,Y 537.764,Z 243.313,A -85,B 0,C 180,E1 -3846.181,E2 -3846.181} C_VEL
LIN {X 0,Y 537.688,Z 247.408,A -85,B 0,C 180,E1 -3848.532,E2 -3848.532} C_VEL
LIN {X 0,Y 537.636,Z 251.618,A -85,B 0,C 180,E1 -3850.925,E2 -3850.925} C_VEL
LIN {X 0,Y 537.604,Z 256.562,A -85,B 0,C 180,E1 -3853.676,E2 -3853.676} C_VEL
LIN {X 0,Y 537.592,Z 257.05,A -85,B 0,C 180,E1 -3853.944,E2 -3853.944} C_VEL
LIN {X 0,Y 540.003,Z 268.992,A -85,B 0,C 180,E1 -3854.264,E2 -3854.264} C_VEL
LIN {X 0,Y 539.793,Z 282.861,A -85,B 0,C 180,E1 -3854.68,E2 -3854.68} C_VEL
LIN {X 0,Y 539.553,Z 295.335,A -85,B 0,C 180,E1 -3855.189,E2 -3855.189} C_VEL
LIN {X 0,Y 539.215,Z 307.994,A -85,B 0,C 180,E1 -3855.855,E2 -3855.855} C_VEL
LIN {X 0,Y 538.902,Z 320.886,A -85,B 0,C 180,E1 -3856.712,E2 -3856.712} C_VEL
LIN {X 0,Y 538.581,Z 332.482,A -85,B 0,C 180,E1 -3857.662,E2 -3857.662} C_VEL
LIN {X 0,Y 538.33,Z 342.973,A -85,B 0,C 180,E1 -3858.707,E2 -3858.707} C_VEL
LIN {X 0,Y 538.06,Z 352.47,A -85,B 0,C 180,E1 -3859.844,E2 -3859.844} C_VEL
LIN {X 0,Y 537.859,Z 361.538,A -85,B 0,C 180,E1 -3861.168,E2 -3861.168} C_VEL
LIN {X 0,Y 537.706,Z 368.838,A -85,B 0,C 180,E1 -3862.49,E2 -3862.49} C_VEL
LIN {X 0,Y 537.645,Z 375.397,A -85,B 0,C 180,E1 -3863.997,E2 -3863.997} C_VEL
LIN {X 0,Y 537.551,Z 380.319,A -85,B 0,C 180,E1 -3865.501,E2 -3865.501} C_VEL
LIN {X 0,Y 537.548,Z 383.749,A -85,B 0,C 180,E1 -3867.002,E2 -3867.002} C_VEL
LIN {X 0,Y 537.449,Z 385.789,A -85,B 0,C 180,E1 -3868.501,E2 -3868.501} C_VEL
LIN {X 0,Y 537.44,Z 386.496,A -85,B 0,C 180,E1 -3870,E2 -3870} C_VEL
LIN {X 0,Y 537.447,Z 385.878,A -85,B 0,C 180,E1 -3871.499,E2 -3871.499} C_VEL
LIN {X 0,Y 537.547,Z 383.918,A -85,B 0,C 180,E1 -3872.998,E2 -3872.998} C_VEL
LIN {X 0,Y 537.551,Z 380.571,A -85,B 0,C 180,E1 -3874.499,E2 -3874.499} C_VEL
LIN {X 0,Y 537.643,Z 375.739,A -85,B 0,C 180,E1 -3876.003,E2 -3876.003} C_VEL
LIN {X 0,Y 537.662,Z 371.078,A -85,B 0,C 180,E1 -3877.133,E2 -3877.133} C_VEL
LIN {X 0,Y 537.824,Z 364.298,A -85,B 0,C 180,E1 -3878.454,E2 -3878.454} C_VEL
LIN {X 0,Y 537.95,Z 355.876,A -85,B 0,C 180,E1 -3879.778,E2 -3879.778} C_VEL
LIN {X 0,Y 538.217,Z 347.089,A -85,B 0,C 180,E1 -3880.914,E2 -3880.914} C_VEL
LIN {X 0,Y 538.468,Z 336.465,A -85,B 0,C 180,E1 -3882.054,E2 -3882.054} C_VEL
LIN {X 0,Y 538.762,Z 325.734,A -85,B 0,C 180,E1 -3883.004,E2 -3883.004} C_VEL
LIN {X 0,Y 539.083,Z 313.992,A -85,B 0,C 180,E1 -3883.86,E2 -3883.86} C_VEL
LIN {X 0,Y 539.401,Z 301.037,A -85,B 0,C 180,E1 -3884.622,E2 -3884.622} C_VEL
LIN {X 0,Y 539.694,Z 287.548,A -85,B 0,C 180,E1 -3885.239,E2 -3885.239} C_VEL
LIN {X 0,Y 539.901,Z 273.868,A -85,B 0,C 180,E1 -3885.7,E2 -3885.7} C_VEL
LIN {X 0,Y 539.875,Z 267.57,A -85,B 0,C 180,E1 -3885.865,E2 -3885.865} C_VEL
LIN {X 0,Y 537.583,Z 257.036,A -85,B 0,C 180,E1 -3886.154,E2 -3886.154} C_VEL
LIN {X 0,Y 537.621,Z 253.185,A -85,B 0,C 180,E1 -3888.285,E2 -3888.285} C_VEL
LIN {X 0,Y 537.628,Z 248.969,A -85,B 0,C 180,E1 -3890.668,E2 -3890.668} C_VEL
LIN {X 0,Y 537.768,Z 243.464,A -85,B 0,C 180,E1 -3893.82,E2 -3893.82} C_VEL
LIN {X 0,Y 537.735,Z 239.073,A -85,B 0,C 180,E1 -3896.383,E2 -3896.383} C_VEL
LIN {X 0,Y 537.862,Z 234.826,A -85,B 0,C 180,E1 -3898.912,E2 -3898.912} C_VEL
LIN {X 0,Y 537.916,Z 229.987,A -85,B 0,C 180,E1 -3901.871,E2 -3901.871} C_VEL
LIN {X 0,Y 538.001,Z 225.606,A -85,B 0,C 180,E1 -3904.615,E2 -3904.615} C_VEL
LIN {X 0,Y 538.076,Z 221.608,A -85,B 0,C 180,E1 -3907.18,E2 -3907.18} C_VEL
LIN {X 0,Y 537.956,Z 219.103,A -85,B 0,C 180,E1 -3908.836,E2 -3908.836} C_VEL
LIN {X 0,Y 538.05,Z 219.089,A -85,B 0,C 180,E1 -3910.776,E2 -3910.776} C_VEL
LIN {X 0,Y 538.007,Z 219.093,A -85,B 0,C 180,E1 -3913.816,E2 -3913.816} C_VEL
LIN {X 0,Y 538.013,Z 219.096,A -85,B 0,C 180,E1 -3916.185,E2 -3916.185} C_VEL
LIN {X 0,Y 538.005,Z 219.095,A -85,B 0,C 180,E1 -3919.259,E2 -3919.259} C_VEL
LIN {X 0,Y 537.993,Z 219.093,A -85,B 0,C 180,E1 -3922.122,E2 -3922.122} C_VEL
LIN {X 0,Y 538.001,Z 219.093,A -85,B 0,C 180,E1 -3924.916,E2 -3924.916} C_VEL
LIN {X 0,Y 538.02,Z 219.096,A -85,B 0,C 180,E1 -3927.617,E2 -3927.617} C_VEL
LIN {X 0,Y 538.008,Z 219.092,A -85,B 0,C 180,E1 -3930.238,E2 -3930.238} C_VEL
LIN {X 0,Y 538.057,Z 219.088,A -85,B 0,C 180,E1 -3932.796,E2 -3932.796} C_VEL
LIN {X 0,Y 538.031,Z 219.088,A -85,B 0,C 180,E1 -3935.292,E2 -3935.292} C_VEL
LIN {X 0,Y 538.018,Z 219.09,A -85,B 0,C 180,E1 -3938.042,E2 -3938.042} C_VEL
LIN {X 0,Y 538.084,Z 219.083,A -85,B 0,C 180,E1 -3940.148,E2 -3940.148} C_VEL
LIN {X 0,Y 538.016,Z 219.091,A -85,B 0,C 180,E1 -3943.299,E2 -3943.299} C_VEL
LIN {X 0,Y 538.065,Z 219.088,A -85,B 0,C 180,E1 -3945.631,E2 -3945.631} C_VEL
LIN {X 0,Y 538.08,Z 219.089,A -85,B 0,C 180,E1 -3948.702,E2 -3948.702} C_VEL
LIN {X 0,Y 538.065,Z 219.088,A -85,B 0,C 180,E1 -3951.739,E2 -3951.739} C_VEL
LIN {X 0,Y 538.124,Z 219.078,A -85,B 0,C 180,E1 -3954.003,E2 -3954.003} C_VEL
LIN {X 0,Y 538.132,Z 219.079,A -85,B 0,C 180,E1 -3957.005,E2 -3957.005} C_VEL
LIN {X 0,Y 538.184,Z 219.07,A -85,B 0,C 180,E1 -3960.748,E2 -3960.748} C_VEL
LIN {X 0,Y 538.141,Z 219.077,A -85,B 0,C 180,E1 -3962.994,E2 -3962.994} C_VEL
LIN {X 0,Y 538.091,Z 219.082,A -85,B 0,C 180,E1 -3965.998,E2 -3965.998} C_VEL
LIN {X 0,Y 538.051,Z 219.086,A -85,B 0,C 180,E1 -3969.018,E2 -3969.018} C_VEL
LIN {X 0,Y 538.087,Z 219.081,A -85,B 0,C 180,E1 -3972.062,E2 -3972.062} C_VEL
LIN {X 0,Y 538.045,Z 219.088,A -85,B 0,C 180,E1 -3975.144,E2 -3975.144} C_VEL
LIN {X 0,Y 538.008,Z 219.093,A -85,B 0,C 180,E1 -3978.271,E2 -3978.271} C_VEL
LIN {X 0,Y 538.04,Z 219.089,A -85,B 0,C 180,E1 -3980.651,E2 -3980.651} C_VEL
LIN {X 0,Y 538.007,Z 219.093,A -85,B 0,C 180,E1 -3983.888,E2 -3983.888} C_VEL
LIN {X 0,Y 538.011,Z 219.093,A -85,B 0,C 180,E1 -3986.368,E2 -3986.368} C_VEL
LIN {X 0,Y 537.994,Z 219.096,A -85,B 0,C 180,E1 -3988.926,E2 -3988.926} C_VEL
LIN {X 0,Y 538.018,Z 219.09,A -85,B 0,C 180,E1 -3991.888,E2 -3991.888} C_VEL
LIN {X 0,Y 538.01,Z 219.093,A -85,B 0,C 180,E1 -3994.617,E2 -3994.617} C_VEL
LIN {X 0,Y 538.001,Z 219.098,A -85,B 0,C 180,E1 -3997.169,E2 -3997.169} C_VEL
LIN {X 0,Y 538.024,Z 219.09,A -85,B 0,C 180,E1 -3999.797,E2 -3999.797} C_VEL
LIN {X 0,Y 538.022,Z 219.092,A -85,B 0,C 180,E1 -4002.786,E2 -4002.786} C_VEL
LIN {X 0,Y 537.999,Z 219.098,A -85,B 0,C 180,E1 -4005.137,E2 -4005.137} C_VEL
LIN {X 0,Y 538.019,Z 219.093,A -85,B 0,C 180,E1 -4008.225,E2 -4008.225} C_VEL
LIN {X 0,Y 538.079,Z 219.211,A -85,B 0,C 180,E1 -4010.025,E2 -4010.025} C_VEL
LIN {X 0,Y 538.44,Z 223.507,A -85,B 0,C 180,E1 -4012.159,E2 -4012.159} C_VEL
LIN {X 0,Y 538.312,Z 229.47,A -85,B 0,C 180,E1 -4014.939,E2 -4014.939} C_VEL
LIN {X 0,Y 538.233,Z 235.475,A -85,B 0,C 180,E1 -4017.632,E2 -4017.632} C_VEL
LIN {X 0,Y 538.117,Z 241.514,A -85,B 0,C 180,E1 -4020.245,E2 -4020.245} C_VEL
LIN {X 0,Y 538.026,Z 248.573,A -85,B 0,C 180,E1 -4023.214,E2 -4023.214} C_VEL
LIN {X 0,Y 537.866,Z 255.758,A -85,B 0,C 180,E1 -4026.156,E2 -4026.156} C_VEL
LIN {X 0,Y 537.801,Z 262.717,A -85,B 0,C 180,E1 -4028.938,E2 -4028.938} C_VEL
LIN {X 0,Y 537.697,Z 269.808,A -85,B 0,C 180,E1 -4031.718,E2 -4031.718} C_VEL
LIN {X 0,Y 537.666,Z 275.55,A -85,B 0,C 180,E1 -4033.891,E2 -4033.891} C_VEL
LIN {X 0,Y 540.015,Z 287.644,A -85,B 0,C 180,E1 -4034.192,E2 -4034.192} C_VEL
LIN {X 0,Y 539.837,Z 301.443,A -85,B 0,C 180,E1 -4034.592,E2 -4034.592} C_VEL
LIN {X 0,Y 539.48,Z 314.068,A -85,B 0,C 180,E1 -4035.091,E2 -4035.091} C_VEL
LIN {X 0,Y 539.2,Z 326.984,A -85,B 0,C 180,E1 -4035.758,E2 -4035.758} C_VEL
LIN {X 0,Y 538.927,Z 338.802,A -85,B 0,C 180,E1 -4036.52,E2 -4036.52} C_VEL
LIN {X 0,Y 538.627,Z 350.807,A -85,B 0,C 180,E1 -4037.472,E2 -4037.472} C_VEL
LIN {X 0,Y 538.389,Z 361.961,A -85,B 0,C 180,E1 -4038.555,E2 -4038.555} C_VEL
LIN {X 0,Y 538.096,Z 371.336,A -85,B 0,C 180,E1 -4039.654,E2 -4039.654} C_VEL
LIN {X 0,Y 537.919,Z 379.404,A -85,B 0,C 180,E1 -4040.79,E2 -4040.79} C_VEL
LIN {X 0,Y 537.763,Z 387.133,A -85,B 0,C 180,E1 -4042.113,E2 -4042.113} C_VEL
LIN {X 0,Y 537.686,Z 393.218,A -85,B 0,C 180,E1 -4043.406,E2 -4043.406} C_VEL
LIN {X 0,Y 537.578,Z 398.2,A -85,B 0,C 180,E1 -4044.749,E2 -4044.749} C_VEL
LIN {X 0,Y 537.576,Z 402.316,A -85,B 0,C 180,E1 -4046.252,E2 -4046.252} C_VEL
LIN {X 0,Y 537.488,Z 405.002,A -85,B 0,C 180,E1 -4047.752,E2 -4047.752} C_VEL
LIN {X 0,Y 537.437,Z 406.334,A -85,B 0,C 180,E1 -4049.251,E2 -4049.251} C_VEL
LIN {X 0,Y 537.437,Z 406.334,A -85,B 0,C 180,E1 -4050.749,E2 -4050.749} C_VEL
LIN {X 0,Y 537.488,Z 405.005,A -85,B 0,C 180,E1 -4052.248,E2 -4052.248} C_VEL
LIN {X 0,Y 537.576,Z 402.32,A -85,B 0,C 180,E1 -4053.748,E2 -4053.748} C_VEL
LIN {X 0,Y 537.578,Z 398.201,A -85,B 0,C 180,E1 -4055.251,E2 -4055.251} C_VEL
LIN {X 0,Y 537.672,Z 393.272,A -85,B 0,C 180,E1 -4056.581,E2 -4056.581} C_VEL
LIN {X 0,Y 537.763,Z 387.134,A -85,B 0,C 180,E1 -4057.887,E2 -4057.887} C_VEL
LIN {X 0,Y 537.918,Z 379.405,A -85,B 0,C 180,E1 -4059.21,E2 -4059.21} C_VEL
LIN {X 0,Y 538.096,Z 371.337,A -85,B 0,C 180,E1 -4060.346,E2 -4060.346} C_VEL
LIN {X 0,Y 538.363,Z 362.034,A -85,B 0,C 180,E1 -4061.438,E2 -4061.438} C_VEL
LIN {X 0,Y 538.627,Z 350.807,A -85,B 0,C 180,E1 -4062.528,E2 -4062.528} C_VEL
LIN {X 0,Y 538.927,Z 338.806,A -85,B 0,C 180,E1 -4063.48,E2 -4063.48} C_VEL
LIN {X 0,Y 539.2,Z 326.989,A -85,B 0,C 180,E1 -4064.242,E2 -4064.242} C_VEL
LIN {X 0,Y 539.489,Z 314.063,A -85,B 0,C 180,E1 -4064.909,E2 -4064.909} C_VEL
LIN {X 0,Y 539.765,Z 300.033,A -85,B 0,C 180,E1 -4065.458,E2 -4065.458} C_VEL
LIN {X 0,Y 539.89,Z 286.436,A -85,B 0,C 180,E1 -4065.838,E2 -4065.838} C_VEL
LIN {X 0,Y 537.642,Z 275.371,A -85,B 0,C 180,E1 -4066.128,E2 -4066.128} C_VEL
LIN {X 0,Y 537.743,Z 267.785,A -85,B 0,C 180,E1 -4069.071,E2 -4069.071} C_VEL
LIN {X 0,Y 537.829,Z 260.58,A -85,B 0,C 180,E1 -4071.908,E2 -4071.908} C_VEL
LIN {X 0,Y 537.903,Z 252.587,A -85,B 0,C 180,E1 -4075.127,E2 -4075.127} C_VEL
LIN {X 0,Y 538.056,Z 245.544,A -85,B 0,C 180,E1 -4078.049,E2 -4078.049} C_VEL
LIN {X 0,Y 538.178,Z 238.49,A -85,B 0,C 180,E1 -4081.053,E2 -4081.053} C_VEL
LIN {X 0,Y 538.309,Z 231.463,A -85,B 0,C 180,E1 -4084.152,E2 -4084.152} C_VEL
LIN {X 0,Y 538.442,Z 224.773,A -85,B 0,C 180,E1 -4087.231,E2 -4087.231} C_VEL
LIN {X 0,Y 538.196,Z 219.931,A -85,B 0,C 180,E1 -4089.606,E2 -4089.606} C_VEL
LIN {X 0,Y 538.05,Z 219.09,A -85,B 0,C 180,E1 -4090.039,E2 -4090.039} C_VEL
LIN {X 0,Y 537.98,Z 219.101,A -85,B 0,C 180,E1 -4092.982,E2 -4092.982} C_VEL
LIN {X 0,Y 538.019,Z 219.095,A -85,B 0,C 180,E1 -4095.927,E2 -4095.927} C_VEL
LIN {X 0,Y 538.038,Z 219.09,A -85,B 0,C 180,E1 -4098.227,E2 -4098.227} C_VEL
LIN {X 0,Y 538.012,Z 219.097,A -85,B 0,C 180,E1 -4101.169,E2 -4101.169} C_VEL
LIN {X 0,Y 537.989,Z 219.098,A -85,B 0,C 180,E1 -4104.09,E2 -4104.09} C_VEL
LIN {X 0,Y 538.032,Z 219.089,A -85,B 0,C 180,E1 -4106.727,E2 -4106.727} C_VEL
LIN {X 0,Y 538.015,Z 219.092,A -85,B 0,C 180,E1 -4109.559,E2 -4109.559} C_VEL
LIN {X 0,Y 537.996,Z 219.094,A -85,B 0,C 180,E1 -4111.948,E2 -4111.948} C_VEL
LIN {X 0,Y 538.049,Z 219.088,A -85,B 0,C 180,E1 -4114.466,E2 -4114.466} C_VEL
LIN {X 0,Y 538.017,Z 219.093,A -85,B 0,C 180,E1 -4116.928,E2 -4116.928} C_VEL
LIN {X 0,Y 538.082,Z 219.084,A -85,B 0,C 180,E1 -4120.148,E2 -4120.148} C_VEL
LIN {X 0,Y 537.988,Z 219.095,A -85,B 0,C 180,E1 -4123.298,E2 -4123.298} C_VEL
LIN {X 0,Y 538.067,Z 219.087,A -85,B 0,C 180,E1 -4125.631,E2 -4125.631} C_VEL
LIN {X 0,Y 538.08,Z 219.086,A -85,B 0,C 180,E1 -4128.702,E2 -4128.702} C_VEL
LIN {X 0,Y 538.041,Z 219.092,A -85,B 0,C 180,E1 -4131.739,E2 -4131.739} C_VEL
LIN {X 0,Y 538.153,Z 219.075,A -85,B 0,C 180,E1 -4134.755,E2 -4134.755} C_VEL
LIN {X 0,Y 538.169,Z 219.072,A -85,B 0,C 180,E1 -4137.755,E2 -4137.755} C_VEL
LIN {X 0,Y 538.176,Z 219.07,A -85,B 0,C 180,E1 -4140.748,E2 -4140.748} C_VEL
LIN {X 0,Y 538.13,Z 219.079,A -85,B 0,C 180,E1 -4142.995,E2 -4142.995} C_VEL
LIN {X 0,Y 538.122,Z 219.078,A -85,B 0,C 180,E1 -4145.997,E2 -4145.997} C_VEL
LIN {X 0,Y 538.063,Z 219.084,A -85,B 0,C 180,E1 -4149.018,E2 -4149.018} C_VEL
LIN {X 0,Y 538.062,Z 219.085,A -85,B 0,C 180,E1 -4152.063,E2 -4152.063} C_VEL
LIN {X 0,Y 538.047,Z 219.087,A -85,B 0,C 180,E1 -4155.144,E2 -4155.144} C_VEL
LIN {X 0,Y 538.031,Z 219.09,A -85,B 0,C 180,E1 -4158.27,E2 -4158.27} C_VEL
LIN {X 0,Y 538.038,Z 219.089,A -85,B 0,C 180,E1 -4160.652,E2 -4160.652} C_VEL
LIN {X 0,Y 538.002,Z 219.093,A -85,B 0,C 180,E1 -4163.889,E2 -4163.889} C_VEL
LIN {X 0,Y 538.042,Z 219.088,A -85,B 0,C 180,E1 -4166.367,E2 -4166.367} C_VEL
LIN {X 0,Y 538.032,Z 219.091,A -85,B 0,C 180,E1 -4168.933,E2 -4168.933} C_VEL
LIN {X 0,Y 538.012,Z 219.092,A -85,B 0,C 180,E1 -4171.887,E2 -4171.887} C_VEL
LIN {X 0,Y 538.012,Z 219.092,A -85,B 0,C 180,E1 -4174.617,E2 -4174.617} C_VEL
LIN {X 0,Y 538.006,Z 219.097,A -85,B 0,C 180,E1 -4177.17,E2 -4177.17} C_VEL
LIN {X 0,Y 538.008,Z 219.091,A -85,B 0,C 180,E1 -4179.799,E2 -4179.799} C_VEL
LIN {X 0,Y 537.988,Z 219.094,A -85,B 0,C 180,E1 -4180.264,E2 -4180.264} C_VEL
LIN {X 0,Y 537.327,Z 219.181,A -85,B 0,C 180,E1 -4180.889,E2 -4180.889} C_VEL
LIN {X 0,Y 534.48,Z 219.539,A -85,B 0,C 180,E1 -4181.904,E2 -4181.904} C_VEL
LIN {X 0,Y 532.068,Z 219.84,A -85,B 0,C 180,E1 -4182.722,E2 -4182.722} C_VEL
LIN {X 0,Y 531.03,Z 219.966,A -85,B 0,C 180,E1 -4183.353,E2 -4183.353} C_VEL
LIN {X 0,Y 530.945,Z 219.974,A -85,B 0,C 180,E1 -4183.566,E2 -4183.566} C_VEL
LIN {X 0,Y 530.956,Z 219.971,A -85,B 0,C 180,E1 -4186.504,E2 -4186.504} C_VEL
LIN {X 0,Y 530.986,Z 219.97,A -85,B 0,C 180,E1 -4188.977,E2 -4188.977} C_VEL
LIN {X 0,Y 530.939,Z 220.177,A -85,B 0,C 180,E1 -4191.351,E2 -4191.351} C_VEL
LIN {X 0,Y 531.01,Z 223.935,A -85,B 0,C 180,E1 -4193.837,E2 -4193.837} C_VEL
LIN {X 0,Y 530.918,Z 228.087,A -85,B 0,C 180,E1 -4196.508,E2 -4196.508} C_VEL
LIN {X 0,Y 530.794,Z 232.683,A -85,B 0,C 180,E1 -4199.388,E2 -4199.388} C_VEL
LIN {X 0,Y 530.708,Z 237.585,A -85,B 0,C 180,E1 -4202.387,E2 -4202.387} C_VEL
LIN {X 0,Y 530.689,Z 241.835,A -85,B 0,C 180,E1 -4204.926,E2 -4204.926} C_VEL
LIN {X 0,Y 530.632,Z 246.086,A -85,B 0,C 180,E1 -4207.413,E2 -4207.413} C_VEL
LIN {X 0,Y 530.579,Z 251.751,A -85,B 0,C 180,E1 -4210.662,E2 -4210.662} C_VEL
LIN {X 0,Y 530.532,Z 257.058,A -85,B 0,C 180,E1 -4213.65,E2 -4213.65} C_VEL
LIN {X 0,Y 530.527,Z 257.204,A -85,B 0,C 180,E1 -4213.732,E2 -4213.732} C_VEL
LIN {X 0,Y 533.171,Z 270.021,A -85,B 0,C 180,E1 -4214.081,E2 -4214.081} C_VEL
LIN {X 0,Y 532.953,Z 283.733,A -85,B 0,C 180,E1 -4214.505,E2 -4214.505} C_VEL
LIN {X 0,Y 532.691,Z 295.482,A -85,B 0,C 180,E1 -4214.994,E2 -4214.994} C_VEL
LIN {X 0,Y 532.33,Z 308.139,A -85,B 0,C 180,E1 -4215.668,E2 -4215.668} C_VEL
LIN {X 0,Y 532.034,Z 319.742,A -85,B 0,C 180,E1 -4216.44,E2 -4216.44} C_VEL
LIN {X 0,Y 531.667,Z 331.558,A -85,B 0,C 180,E1 -4217.402,E2 -4217.402} C_VEL
LIN {X 0,Y 531.38,Z 342.075,A -85,B 0,C 180,E1 -4218.444,E2 -4218.444} C_VEL
LIN {X 0,Y 531.095,Z 351.099,A -85,B 0,C 180,E1 -4219.516,E2 -4219.516} C_VEL
LIN {X 0,Y 530.888,Z 359.194,A -85,B 0,C 180,E1 -4220.667,E2 -4220.667} C_VEL
LIN {X 0,Y 530.705,Z 366.943,A -85,B 0,C 180,E1 -4222.007,E2 -4222.007} C_VEL
LIN {X 0,Y 530.575,Z 373.562,A -85,B 0,C 180,E1 -4223.44,E2 -4223.44} C_VEL
LIN {X 0,Y 530.514,Z 378.055,A -85,B 0,C 180,E1 -4224.679,E2 -4224.679} C_VEL
LIN {X 0,Y 530.497,Z 382.214,A -85,B 0,C 180,E1 -4226.202,E2 -4226.202} C_VEL
LIN {X 0,Y 530.409,Z 384.939,A -85,B 0,C 180,E1 -4227.722,E2 -4227.722} C_VEL
LIN {X 0,Y 530.34,Z 386.309,A -85,B 0,C 180,E1 -4229.241,E2 -4229.241} C_VEL
LIN {X 0,Y 530.342,Z 386.353,A -85,B 0,C 180,E1 -4230.759,E2 -4230.759} C_VEL
LIN {X 0,Y 530.408,Z 385.067,A -85,B 0,C 180,E1 -4232.278,E2 -4232.278} C_VEL
LIN {X 0,Y 530.497,Z 382.421,A -85,B 0,C 180,E1 -4233.798,E2 -4233.798} C_VEL
LIN {X 0,Y 530.514,Z 378.347,A -85,B 0,C 180,E1 -4235.321,E2 -4235.321} C_VEL
LIN {X 0,Y 530.575,Z 372.737,A -85,B 0,C 180,E1 -4236.847,E2 -4236.847} C_VEL
LIN {X 0,Y 530.696,Z 366.41,A -85,B 0,C 180,E1 -4238.185,E2 -4238.185} C_VEL
LIN {X 0,Y 530.909,Z 358.541,A -85,B 0,C 180,E1 -4239.525,E2 -4239.525} C_VEL
LIN {X 0,Y 531.116,Z 350.309,A -85,B 0,C 180,E1 -4240.676,E2 -4240.676} C_VEL
LIN {X 0,Y 531.455,Z 339.918,A -85,B 0,C 180,E1 -4241.879,E2 -4241.879} C_VEL
LIN {X 0,Y 531.743,Z 329.346,A -85,B 0,C 180,E1 -4242.888,E2 -4242.888} C_VEL
LIN {X 0,Y 532.051,Z 318.352,A -85,B 0,C 180,E1 -4243.755,E2 -4243.755} C_VEL
LIN {X 0,Y 532.387,Z 306.424,A -85,B 0,C 180,E1 -4244.526,E2 -4244.526} C_VEL
LIN {X 0,Y 532.676,Z 293.256,A -85,B 0,C 180,E1 -4245.202,E2 -4245.202} C_VEL
LIN {X 0,Y 532.98,Z 279.039,A -85,B 0,C 180,E1 -4245.75,E2 -4245.75} C_VEL
LIN {X 0,Y 533.034,Z 268.592,A -85,B 0,C 180,E1 -4246.052,E2 -4246.052} C_VEL
LIN {X 0,Y 530.547,Z 257.174,A -85,B 0,C 180,E1 -4246.374,E2 -4246.374} C_VEL
LIN {X 0,Y 530.579,Z 251.909,A -85,B 0,C 180,E1 -4249.339,E2 -4249.339} C_VEL
LIN {X 0,Y 530.632,Z 246.24,A -85,B 0,C 180,E1 -4252.588,E2 -4252.588} C_VEL
LIN {X 0,Y 530.692,Z 241.984,A -85,B 0,C 180,E1 -4255.074,E2 -4255.074} C_VEL
LIN {X 0,Y 530.754,Z 236.318,A -85,B 0,C 180,E1 -4258.47,E2 -4258.47} C_VEL
LIN {X 0,Y 530.813,Z 232.062,A -85,B 0,C 180,E1 -4261.089,E2 -4261.089} C_VEL
LIN {X 0,Y 530.905,Z 227.786,A -85,B 0,C 180,E1 -4263.779,E2 -4263.779} C_VEL
LIN {X 0,Y 530.999,Z 223.484,A -85,B 0,C 180,E1 -4266.555,E2 -4266.555} C_VEL
LIN {X 0,Y 530.936,Z 220.32,A -85,B 0,C 180,E1 -4268.649,E2 -4268.649} C_VEL
LIN {X 0,Y 530.975,Z 219.971,A -85,B 0,C 180,E1 -4270.434,E2 -4270.434} C_VEL
LIN {X 0,Y 530.964,Z 219.974,A -85,B 0,C 180,E1 -4273.281,E2 -4273.281} C_VEL
LIN {X 0,Y 530.983,Z 219.968,A -85,B 0,C 180,E1 -4275.622,E2 -4275.622} C_VEL
LIN {X 0,Y 530.966,Z 219.97,A -85,B 0,C 180,E1 -4278.562,E2 -4278.562} C_VEL
LIN {X 0,Y 530.957,Z 219.972,A -85,B 0,C 180,E1 -4281.529,E2 -4281.529} C_VEL
LIN {X 0,Y 530.957,Z 219.976,A -85,B 0,C 180,E1 -4284.38,E2 -4284.38} C_VEL
LIN {X 0,Y 530.97,Z 219.969,A -85,B 0,C 180,E1 -4287.133,E2 -4287.133} C_VEL
LIN {X 0,Y 530.953,Z 219.971,A -85,B 0,C 180,E1 -4289.802,E2 -4289.802} C_VEL
LIN {X 0,Y 531.014,Z 219.969,A -85,B 0,C 180,E1 -4292.468,E2 -4292.468} C_VEL
LIN {X 0,Y 530.998,Z 219.963,A -85,B 0,C 180,E1 -4294.942,E2 -4294.942} C_VEL
LIN {X 0,Y 530.974,Z 219.967,A -85,B 0,C 180,E1 -4298.247,E2 -4298.247} C_VEL
LIN {X 0,Y 530.988,Z 219.971,A -85,B 0,C 180,E1 -4300.677,E2 -4300.677} C_VEL
LIN {X 0,Y 530.974,Z 219.968,A -85,B 0,C 180,E1 -4303.07,E2 -4303.07} C_VEL
LIN {X 0,Y 531.022,Z 219.967,A -85,B 0,C 180,E1 -4305.436,E2 -4305.436} C_VEL
LIN {X 0,Y 531.038,Z 219.964,A -85,B 0,C 180,E1 -4308.55,E2 -4308.55} C_VEL
LIN {X 0,Y 531.04,Z 219.962,A -85,B 0,C 180,E1 -4311.629,E2 -4311.629} C_VEL
LIN {X 0,Y 531.122,Z 219.949,A -85,B 0,C 180,E1 -4314.685,E2 -4314.685} C_VEL
LIN {X 0,Y 531.131,Z 219.948,A -85,B 0,C 180,E1 -4317.725,E2 -4317.725} C_VEL
LIN {X 0,Y 531.155,Z 219.945,A -85,B 0,C 180,E1 -4320.758,E2 -4320.758} C_VEL
LIN {X 0,Y 531.108,Z 219.953,A -85,B 0,C 180,E1 -4323.034,E2 -4323.034} C_VEL
LIN {X 0,Y 531.05,Z 219.959,A -85,B 0,C 180,E1 -4326.077,E2 -4326.077} C_VEL
LIN {X 0,Y 531.014,Z 219.963,A -85,B 0,C 180,E1 -4329.138,E2 -4329.138} C_VEL
LIN {X 0,Y 531.044,Z 219.958,A -85,B 0,C 180,E1 -4332.225,E2 -4332.225} C_VEL
LIN {X 0,Y 530.989,Z 219.966,A -85,B 0,C 180,E1 -4335.35,E2 -4335.35} C_VEL
LIN {X 0,Y 530.971,Z 219.968,A -85,B 0,C 180,E1 -4338.522,E2 -4338.522} C_VEL
LIN {X 0,Y 531.002,Z 219.968,A -85,B 0,C 180,E1 -4340.938,E2 -4340.938} C_VEL
LIN {X 0,Y 530.966,Z 219.973,A -85,B 0,C 180,E1 -4344.225,E2 -4344.225} C_VEL
LIN {X 0,Y 530.962,Z 219.969,A -85,B 0,C 180,E1 -4346.746,E2 -4346.746} C_VEL
LIN {X 0,Y 530.964,Z 219.974,A -85,B 0,C 180,E1 -4349.324,E2 -4349.324} C_VEL
LIN {X 0,Y 530.974,Z 219.969,A -85,B 0,C 180,E1 -4352.101,E2 -4352.101} C_VEL
LIN {X 0,Y 530.968,Z 219.969,A -85,B 0,C 180,E1 -4354.85,E2 -4354.85} C_VEL
LIN {X 0,Y 530.965,Z 219.974,A -85,B 0,C 180,E1 -4357.508,E2 -4357.508} C_VEL
LIN {X 0,Y 530.984,Z 219.972,A -85,B 0,C 180,E1 -4360.433,E2 -4360.433} C_VEL
LIN {X 0,Y 530.963,Z 219.972,A -85,B 0,C 180,E1 -4363.281,E2 -4363.281} C_VEL
LIN {X 0,Y 530.968,Z 219.974,A -85,B 0,C 180,E1 -4365.623,E2 -4365.623} C_VEL
LIN {X 0,Y 530.987,Z 219.971,A -85,B 0,C 180,E1 -4368.563,E2 -4368.563} C_VEL
LIN {X 0,Y 531.04,Z 220.161,A -85,B 0,C 180,E1 -4369.882,E2 -4369.882} C_VEL
LIN {X 0,Y 531.409,Z 223.472,A -85,B 0,C 180,E1 -4371.568,E2 -4371.568} C_VEL
LIN {X 0,Y 531.367,Z 228.088,A -85,B 0,C 180,E1 -4373.785,E2 -4373.785} C_VEL
LIN {X 0,Y 531.281,Z 233.86,A -85,B 0,C 180,E1 -4376.449,E2 -4376.449} C_VEL
LIN {X 0,Y 531.145,Z 240.323,A -85,B 0,C 180,E1 -4379.324,E2 -4379.324} C_VEL
LIN {X 0,Y 531.011,Z 247.638,A -85,B 0,C 180,E1 -4382.468,E2 -4382.468} C_VEL
LIN {X 0,Y 530.852,Z 254.543,A -85,B 0,C 180,E1 -4385.353,E2 -4385.353} C_VEL
LIN {X 0,Y 530.738,Z 262.63,A -85,B 0,C 180,E1 -4388.644,E2 -4388.644} C_VEL
LIN {X 0,Y 530.621,Z 269.723,A -85,B 0,C 180,E1 -4391.465,E2 -4391.465} C_VEL
LIN {X 0,Y 530.571,Z 275.409,A -85,B 0,C 180,E1 -4393.67,E2 -4393.67} C_VEL
LIN {X 0,Y 533.162,Z 288.758,A -85,B 0,C 180,E1 -4394.016,E2 -4394.016} C_VEL
LIN {X 0,Y 532.974,Z 301.833,A -85,B 0,C 180,E1 -4394.408,E2 -4394.408} C_VEL
LIN {X 0,Y 532.545,Z 315.924,A -85,B 0,C 180,E1 -4394.99,E2 -4394.99} C_VEL
LIN {X 0,Y 532.235,Z 328.433,A -85,B 0,C 180,E1 -4395.665,E2 -4395.665} C_VEL
LIN {X 0,Y 531.901,Z 341.255,A -85,B 0,C 180,E1 -4396.533,E2 -4396.533} C_VEL
LIN {X 0,Y 531.584,Z 352.815,A -85,B 0,C 180,E1 -4397.497,E2 -4397.497} C_VEL
LIN {X 0,Y 531.322,Z 363.29,A -85,B 0,C 180,E1 -4398.556,E2 -4398.556} C_VEL
LIN {X 0,Y 531.023,Z 372.753,A -85,B 0,C 180,E1 -4399.708,E2 -4399.708} C_VEL
LIN {X 0,Y 530.818,Z 381.769,A -85,B 0,C 180,E1 -4401.05,E2 -4401.05} C_VEL
LIN {X 0,Y 530.641,Z 389.052,A -85,B 0,C 180,E1 -4402.389,E2 -4402.389} C_VEL
LIN {X 0,Y 530.557,Z 395.568,A -85,B 0,C 180,E1 -4403.917,E2 -4403.917} C_VEL
LIN {X 0,Y 530.449,Z 400.443,A -85,B 0,C 180,E1 -4405.44,E2 -4405.44} C_VEL
LIN {X 0,Y 530.452,Z 403.832,A -85,B 0,C 180,E1 -4406.962,E2 -4406.962} C_VEL
LIN {X 0,Y 530.357,Z 405.835,A -85,B 0,C 180,E1 -4408.481,E2 -4408.481} C_VEL
LIN {X 0,Y 530.341,Z 406.5,A -85,B 0,C 180,E1 -4410,E2 -4410} C_VEL
LIN {X 0,Y 530.357,Z 405.837,A -85,B 0,C 180,E1 -4411.519,E2 -4411.519} C_VEL
LIN {X 0,Y 530.452,Z 403.836,A -85,B 0,C 180,E1 -4413.038,E2 -4413.038} C_VEL
LIN {X 0,Y 530.449,Z 400.447,A -85,B 0,C 180,E1 -4414.559,E2 -4414.559} C_VEL
LIN {X 0,Y 530.546,Z 395.567,A -85,B 0,C 180,E1 -4416.083,E2 -4416.083} C_VEL
LIN {X 0,Y 530.641,Z 389.052,A -85,B 0,C 180,E1 -4417.611,E2 -4417.611} C_VEL
LIN {X 0,Y 530.818,Z 381.771,A -85,B 0,C 180,E1 -4418.95,E2 -4418.95} C_VEL
LIN {X 0,Y 531.023,Z 372.754,A -85,B 0,C 180,E1 -4420.292,E2 -4420.292} C_VEL
LIN {X 0,Y 531.315,Z 363.291,A -85,B 0,C 180,E1 -4421.444,E2 -4421.444} C_VEL
LIN {X 0,Y 531.584,Z 352.816,A -85,B 0,C 180,E1 -4422.503,E2 -4422.503} C_VEL
LIN {X 0,Y 531.901,Z 341.259,A -85,B 0,C 180,E1 -4423.467,E2 -4423.467} C_VEL
LIN {X 0,Y 532.234,Z 328.439,A -85,B 0,C 180,E1 -4424.335,E2 -4424.335} C_VEL
LIN {X 0,Y 532.552,Z 315.92,A -85,B 0,C 180,E1 -4425.01,E2 -4425.01} C_VEL
LIN {X 0,Y 532.913,Z 303.206,A -85,B 0,C 180,E1 -4425.542,E2 -4425.542} C_VEL
LIN {X 0,Y 533.142,Z 289.576,A -85,B 0,C 180,E1 -4425.962,E2 -4425.962} C_VEL
LIN {X 0,Y 532.691,Z 285.656,A -85,B 0,C 180,E1 -4426.071,E2 -4426.071} C_VEL
LIN {X 0,Y 530.565,Z 275.251,A -85,B 0,C 180,E1 -4426.349,E2 -4426.349} C_VEL
LIN {X 0,Y 530.67,Z 267.7,A -85,B 0,C 180,E1 -4429.335,E2 -4429.335} C_VEL
LIN {X 0,Y 530.755,Z 260.923,A -85,B 0,C 180,E1 -4432.042,E2 -4432.042} C_VEL
LIN {X 0,Y 530.842,Z 253.526,A -85,B 0,C 180,E1 -4435.066,E2 -4435.066} C_VEL
LIN {X 0,Y 531.03,Z 246.479,A -85,B 0,C 180,E1 -4438.023,E2 -4438.023} C_VEL
LIN {X 0,Y 531.141,Z 239.431,A -85,B 0,C 180,E1 -4441.067,E2 -4441.067} C_VEL
LIN {X 0,Y 531.283,Z 233.406,A -85,B 0,C 180,E1 -4443.751,E2 -4443.751} C_VEL
LIN {X 0,Y 531.369,Z 227.422,A -85,B 0,C 180,E1 -4446.526,E2 -4446.526} C_VEL
LIN {X 0,Y 531.36,Z 222.918,A -85,B 0,C 180,E1 -4448.706,E2 -4448.706} C_VEL
LIN {X 0,Y 531.02,Z 219.966,A -85,B 0,C 180,E1 -4450.274,E2 -4450.274} C_VEL
LIN {X 0,Y 530.938,Z 219.975,A -85,B 0,C 180,E1 -4453.498,E2 -4453.498} C_VEL
LIN {X 0,Y 530.955,Z 219.974,A -85,B 0,C 180,E1 -4456.504,E2 -4456.504} C_VEL
LIN {X 0,Y 530.987,Z 219.968,A -85,B 0,C 180,E1 -4458.976,E2 -4458.976} C_VEL
LIN {X 0,Y 530.955,Z 219.972,A -85,B 0,C 180,E1 -4461.529,E2 -4461.529} C_VEL
LIN {X 0,Y 530.949,Z 219.977,A -85,B 0,C 180,E1 -4464.38,E2 -4464.38} C_VEL
LIN {X 0,Y 530.972,Z 219.97,A -85,B 0,C 180,E1 -4467.134,E2 -4467.134} C_VEL
LIN {X 0,Y 530.96,Z 219.97,A -85,B 0,C 180,E1 -4469.802,E2 -4469.802} C_VEL
LIN {X 0,Y 530.965,Z 219.974,A -85,B 0,C 180,E1 -4472.478,E2 -4472.478} C_VEL
LIN {X 0,Y 530.981,Z 219.967,A -85,B 0,C 180,E1 -4474.941,E2 -4474.941} C_VEL
LIN {X 0,Y 530.974,Z 219.968,A -85,B 0,C 180,E1 -4478.247,E2 -4478.247} C_VEL
LIN {X 0,Y 530.982,Z 219.971,A -85,B 0,C 180,E1 -4480.677,E2 -4480.677} C_VEL
LIN {X 0,Y 530.955,Z 219.97,A -85,B 0,C 180,E1 -4483.07,E2 -4483.07} C_VEL
LIN {X 0,Y 531.044,Z 219.963,A -85,B 0,C 180,E1 -4485.437,E2 -4485.437} C_VEL
LIN {X 0,Y 531.04,Z 219.965,A -85,B 0,C 180,E1 -4488.55,E2 -4488.55} C_VEL
LIN {X 0,Y 530.992,Z 219.968,A -85,B 0,C 180,E1 -4491.628,E2 -4491.628} C_VEL
LIN {X 0,Y 531.11,Z 219.952,A -85,B 0,C 180,E1 -4494.685,E2 -4494.685} C_VEL
LIN {X 0,Y 531.141,Z 219.947,A -85,B 0,C 180,E1 -4497.725,E2 -4497.725} C_VEL
LIN {X 0,Y 531.148,Z 219.946,A -85,B 0,C 180,E1 -4500.758,E2 -4500.758} C_VEL
LIN {X 0,Y 531.097,Z 219.956,A -85,B 0,C 180,E1 -4503.034,E2 -4503.034} C_VEL
LIN {X 0,Y 531.078,Z 219.956,A -85,B 0,C 180,E1 -4506.077,E2 -4506.077} C_VEL
LIN {X 0,Y 531.056,Z 219.96,A -85,B 0,C 180,E1 -4508.371,E2 -4508.371} C_VEL
LIN {X 0,Y 531.052,Z 219.96,A -85,B 0,C 180,E1 -4511.671,E2 -4511.671} C_VEL
LIN {X 0,Y 531.031,Z 219.962,A -85,B 0,C 180,E1 -4514.955,E2 -4514.955} C_VEL
LIN {X 0,Y 531.019,Z 219.967,A -85,B 0,C 180,E1 -4517.722,E2 -4517.722} C_VEL
LIN {X 0,Y 531.027,Z 219.961,A -85,B 0,C 180,E1 -4520.127,E2 -4520.127} C_VEL
LIN {X 0,Y 530.945,Z 219.976,A -85,B 0,C 180,E1 -4522.574,E2 -4522.574} C_VEL
LIN {X 0,Y 530.996,Z 219.965,A -85,B 0,C 180,E1 -4525.058,E2 -4525.058} C_VEL
LIN {X 0,Y 531.011,Z 219.968,A -85,B 0,C 180,E1 -4527.596,E2 -4527.596} C_VEL
LIN {X 0,Y 530.967,Z 219.973,A -85,B 0,C 180,E1 -4530.643,E2 -4530.643} C_VEL
LIN {X 0,Y 530.965,Z 219.969,A -85,B 0,C 180,E1 -4533.5,E2 -4533.5} C_VEL
LIN {X 0,Y 530.947,Z 219.972,A -85,B 0,C 180,E1 -4536.153,E2 -4536.153} C_VEL
LIN {X 0,Y 530.966,Z 219.972,A -85,B 0,C 180,E1 -4538.653,E2 -4538.653} C_VEL
LIN {X 0,Y 530.965,Z 219.969,A -85,B 0,C 180,E1 -4541.439,E2 -4541.439} C_VEL
LIN {X 0,Y 530.945,Z 219.974,A -85,B 0,C 180,E1 -4543.566,E2 -4543.566} C_VEL
LIN {X 0,Y 530.277,Z 220.057,A -85,B 0,C 180,E1 -4544.2,E2 -4544.2} C_VEL
LIN {X 0,Y 527.434,Z 220.413,A -85,B 0,C 180,E1 -4545.229,E2 -4545.229} C_VEL
LIN {X 0,Y 525.032,Z 220.715,A -85,B 0,C 180,E1 -4546.058,E2 -4546.058} C_VEL
LIN {X 0,Y 524.001,Z 220.842,A -85,B 0,C 180,E1 -4546.697,E2 -4546.697} C_VEL
LIN {X 0,Y 523.917,Z 220.851,A -85,B 0,C 180,E1 -4546.914,E2 -4546.914} C_VEL
LIN {X 0,Y 523.941,Z 220.848,A -85,B 0,C 180,E1 -4548.908,E2 -4548.908} C_VEL
LIN {X 0,Y 523.896,Z 220.853,A -85,B 0,C 180,E1 -4551.084,E2 -4551.084} C_VEL
LIN {X 0,Y 523.958,Z 224.466,A -85,B 0,C 180,E1 -4553.591,E2 -4553.591} C_VEL
LIN {X 0,Y 523.855,Z 229.129,A -85,B 0,C 180,E1 -4556.629,E2 -4556.629} C_VEL
LIN {X 0,Y 523.752,Z 233.408,A -85,B 0,C 180,E1 -4559.342,E2 -4559.342} C_VEL
LIN {X 0,Y 523.65,Z 238.261,A -85,B 0,C 180,E1 -4562.35,E2 -4562.35} C_VEL
LIN {X 0,Y 523.621,Z 241.911,A -85,B 0,C 180,E1 -4564.564,E2 -4564.564} C_VEL
LIN {X 0,Y 523.572,Z 246.166,A -85,B 0,C 180,E1 -4567.091,E2 -4567.091} C_VEL
LIN {X 0,Y 523.519,Z 251.894,A -85,B 0,C 180,E1 -4570.39,E2 -4570.39} C_VEL
LIN {X 0,Y 523.466,Z 257.337,A -85,B 0,C 180,E1 -4573.501,E2 -4573.501} C_VEL
LIN {X 0,Y 526.34,Z 271.087,A -85,B 0,C 180,E1 -4573.893,E2 -4573.893} C_VEL
LIN {X 0,Y 526.112,Z 284.434,A -85,B 0,C 180,E1 -4574.32,E2 -4574.32} C_VEL
LIN {X 0,Y 525.759,Z 297.615,A -85,B 0,C 180,E1 -4574.891,E2 -4574.891} C_VEL
LIN {X 0,Y 525.387,Z 309.862,A -85,B 0,C 180,E1 -4575.573,E2 -4575.573} C_VEL
LIN {X 0,Y 525.013,Z 322.46,A -85,B 0,C 180,E1 -4576.452,E2 -4576.452} C_VEL
LIN {X 0,Y 524.643,Z 333.832,A -85,B 0,C 180,E1 -4577.427,E2 -4577.427} C_VEL
LIN {X 0,Y 524.366,Z 343.254,A -85,B 0,C 180,E1 -4578.402,E2 -4578.402} C_VEL
LIN {X 0,Y 524.017,Z 352.719,A -85,B 0,C 180,E1 -4579.569,E2 -4579.569} C_VEL
LIN {X 0,Y 523.778,Z 361.749,A -85,B 0,C 180,E1 -4580.929,E2 -4580.929} C_VEL
LIN {X 0,Y 523.598,Z 369.017,A -85,B 0,C 180,E1 -4582.286,E2 -4582.286} C_VEL
LIN {X 0,Y 523.489,Z 375.544,A -85,B 0,C 180,E1 -4583.834,E2 -4583.834} C_VEL
LIN {X 0,Y 523.355,Z 380.442,A -85,B 0,C 180,E1 -4585.379,E2 -4585.379} C_VEL
LIN {X 0,Y 523.419,Z 382.324,A -85,B 0,C 180,E1 -4586.151,E2 -4586.151} C_VEL
LIN {X 0,Y 523.333,Z 385.035,A -85,B 0,C 180,E1 -4587.691,E2 -4587.691} C_VEL
LIN {X 0,Y 523.246,Z 386.399,A -85,B 0,C 180,E1 -4589.23,E2 -4589.23} C_VEL
LIN {X 0,Y 523.248,Z 386.442,A -85,B 0,C 180,E1 -4590.77,E2 -4590.77} C_VEL
LIN {X 0,Y 523.332,Z 385.161,A -85,B 0,C 180,E1 -4592.309,E2 -4592.309} C_VEL
LIN {X 0,Y 523.419,Z 382.527,A -85,B 0,C 180,E1 -4593.85,E2 -4593.85} C_VEL
LIN {X 0,Y 523.448,Z 378.473,A -85,B 0,C 180,E1 -4595.393,E2 -4595.393} C_VEL
LIN {X 0,Y 523.496,Z 372.87,A -85,B 0,C 180,E1 -4596.94,E2 -4596.94} C_VEL
LIN {X 0,Y 523.654,Z 366.542,A -85,B 0,C 180,E1 -4598.295,E2 -4598.295} C_VEL
LIN {X 0,Y 523.872,Z 358.672,A -85,B 0,C 180,E1 -4599.654,E2 -4599.654} C_VEL
LIN {X 0,Y 524.116,Z 350.439,A -85,B 0,C 180,E1 -4600.82,E2 -4600.82} C_VEL
LIN {X 0,Y 524.44,Z 340.726,A -85,B 0,C 180,E1 -4601.966,E2 -4601.966} C_VEL
LIN {X 0,Y 524.783,Z 329.475,A -85,B 0,C 180,E1 -4603.061,E2 -4603.061} C_VEL
LIN {X 0,Y 525.145,Z 318.479,A -85,B 0,C 180,E1 -4603.939,E2 -4603.939} C_VEL
LIN {X 0,Y 525.519,Z 306.548,A -85,B 0,C 180,E1 -4604.72,E2 -4604.72} C_VEL
LIN {X 0,Y 525.836,Z 293.376,A -85,B 0,C 180,E1 -4605.405,E2 -4605.405} C_VEL
LIN {X 0,Y 526.143,Z 279.182,A -85,B 0,C 180,E1 -4605.959,E2 -4605.959} C_VEL
LIN {X 0,Y 526.167,Z 269.452,A -85,B 0,C 180,E1 -4606.247,E2 -4606.247} C_VEL
LIN {X 0,Y 523.456,Z 257.313,A -85,B 0,C 180,E1 -4606.602,E2 -4606.602} C_VEL
LIN {X 0,Y 523.519,Z 252.049,A -85,B 0,C 180,E1 -4609.61,E2 -4609.61} C_VEL
LIN {X 0,Y 523.573,Z 246.317,A -85,B 0,C 180,E1 -4612.909,E2 -4612.909} C_VEL
LIN {X 0,Y 523.623,Z 242.062,A -85,B 0,C 180,E1 -4615.436,E2 -4615.436} C_VEL
LIN {X 0,Y 523.728,Z 236.395,A -85,B 0,C 180,E1 -4618.888,E2 -4618.888} C_VEL
LIN {X 0,Y 523.774,Z 232.13,A -85,B 0,C 180,E1 -4621.554,E2 -4621.554} C_VEL
LIN {X 0,Y 523.899,Z 227.847,A -85,B 0,C 180,E1 -4624.293,E2 -4624.293} C_VEL
LIN {X 0,Y 523.956,Z 223.53,A -85,B 0,C 180,E1 -4627.128,E2 -4627.128} C_VEL
LIN {X 0,Y 523.866,Z 220.886,A -85,B 0,C 180,E1 -4628.912,E2 -4628.912} C_VEL
LIN {X 0,Y 523.958,Z 220.848,A -85,B 0,C 180,E1 -4631.31,E2 -4631.31} C_VEL
LIN {X 0,Y 523.953,Z 220.849,A -85,B 0,C 180,E1 -4634.691,E2 -4634.691} C_VEL
LIN {X 0,Y 523.934,Z 220.851,A -85,B 0,C 180,E1 -4637.879,E2 -4637.879} C_VEL
LIN {X 0,Y 523.915,Z 220.852,A -85,B 0,C 180,E1 -4641.081,E2 -4641.081} C_VEL
LIN {X 0,Y 523.903,Z 220.849,A -85,B 0,C 180,E1 -4643.825,E2 -4643.825} C_VEL
LIN {X 0,Y 523.916,Z 220.847,A -85,B 0,C 180,E1 -4646.634,E2 -4646.634} C_VEL
LIN {X 0,Y 523.944,Z 220.849,A -85,B 0,C 180,E1 -4649.355,E2 -4649.355} C_VEL
LIN {X 0,Y 523.977,Z 220.843,A -85,B 0,C 180,E1 -4652.282,E2 -4652.282} C_VEL
LIN {X 0,Y 523.951,Z 220.842,A -85,B 0,C 180,E1 -4654.581,E2 -4654.581} C_VEL
LIN {X 0,Y 523.921,Z 220.848,A -85,B 0,C 180,E1 -4657.757,E2 -4657.757} C_VEL
LIN {X 0,Y 523.973,Z 220.843,A -85,B 0,C 180,E1 -4660.408,E2 -4660.408} C_VEL
LIN {X 0,Y 523.95,Z 220.843,A -85,B 0,C 180,E1 -4662.837,E2 -4662.837} C_VEL
LIN {X 0,Y 523.98,Z 220.842,A -85,B 0,C 180,E1 -4665.236,E2 -4665.236} C_VEL
LIN {X 0,Y 524.017,Z 220.837,A -85,B 0,C 180,E1 -4668.394,E2 -4668.394} C_VEL
LIN {X 0,Y 523.991,Z 220.839,A -85,B 0,C 180,E1 -4671.516,E2 -4671.516} C_VEL
LIN {X 0,Y 524.041,Z 220.834,A -85,B 0,C 180,E1 -4673.841,E2 -4673.841} C_VEL
LIN {X 0,Y 524.041,Z 220.836,A -85,B 0,C 180,E1 -4676.925,E2 -4676.925} C_VEL
LIN {X 0,Y 524.103,Z 220.829,A -85,B 0,C 180,E1 -4680,E2 -4680} C_VEL
LIN {X 0,Y 524.074,Z 220.83,A -85,B 0,C 180,E1 -4683.075,E2 -4683.075} C_VEL
LIN {X 0,Y 524.011,Z 220.837,A -85,B 0,C 180,E1 -4686.159,E2 -4686.159} C_VEL
LIN {X 0,Y 523.984,Z 220.839,A -85,B 0,C 180,E1 -4689.262,E2 -4689.262} C_VEL
LIN {X 0,Y 524.007,Z 220.837,A -85,B 0,C 180,E1 -4691.739,E2 -4691.739} C_VEL
LIN {X 0,Y 523.998,Z 220.838,A -85,B 0,C 180,E1 -4695.053,E2 -4695.053} C_VEL
LIN {X 0,Y 523.918,Z 220.852,A -85,B 0,C 180,E1 -4697.971,E2 -4697.971} C_VEL
LIN {X 0,Y 523.975,Z 220.84,A -85,B 0,C 180,E1 -4700.41,E2 -4700.41} C_VEL
LIN {X 0,Y 523.915,Z 220.851,A -85,B 0,C 180,E1 -4702.893,E2 -4702.893} C_VEL
LIN {X 0,Y 523.923,Z 220.846,A -85,B 0,C 180,E1 -4705.42,E2 -4705.42} C_VEL
LIN {X 0,Y 523.91,Z 220.849,A -85,B 0,C 180,E1 -4708.002,E2 -4708.002} C_VEL
LIN {X 0,Y 523.94,Z 220.849,A -85,B 0,C 180,E1 -4710.853,E2 -4710.853} C_VEL
LIN {X 0,Y 523.961,Z 220.843,A -85,B 0,C 180,E1 -4713.734,E2 -4713.734} C_VEL
LIN {X 0,Y 523.899,Z 220.85,A -85,B 0,C 180,E1 -4716.4,E2 -4716.4} C_VEL
LIN {X 0,Y 523.921,Z 220.851,A -85,B 0,C 180,E1 -4719.085,E2 -4719.085} C_VEL
LIN {X 0,Y 523.957,Z 220.848,A -85,B 0,C 180,E1 -4722.119,E2 -4722.119} C_VEL
LIN {X 0,Y 523.938,Z 220.851,A -85,B 0,C 180,E1 -4725.311,E2 -4725.311} C_VEL
LIN {X 0,Y 523.951,Z 220.848,A -85,B 0,C 180,E1 -4728.69,E2 -4728.69} C_VEL
LIN {X 0,Y 524.005,Z 220.99,A -85,B 0,C 180,E1 -4729.674,E2 -4729.674} C_VEL
LIN {X 0,Y 524.413,Z 225.405,A -85,B 0,C 180,E1 -4731.941,E2 -4731.941} C_VEL
LIN {X 0,Y 524.307,Z 231.473,A -85,B 0,C 180,E1 -4734.852,E2 -4734.852} C_VEL
LIN {X 0,Y 524.172,Z 237.523,A -85,B 0,C 180,E1 -4737.639,E2 -4737.639} C_VEL
LIN {X 0,Y 524.053,Z 243.386,A -85,B 0,C 180,E1 -4740.251,E2 -4740.251} C_VEL
LIN {X 0,Y 523.927,Z 250.434,A -85,B 0,C 180,E1 -4743.296,E2 -4743.296} C_VEL
LIN {X 0,Y 523.731,Z 257.485,A -85,B 0,C 180,E1 -4746.261,E2 -4746.261} C_VEL
LIN {X 0,Y 523.666,Z 264.572,A -85,B 0,C 180,E1 -4749.167,E2 -4749.167} C_VEL
LIN {X 0,Y 523.545,Z 271.612,A -85,B 0,C 180,E1 -4752.016,E2 -4752.016} C_VEL
LIN {X 0,Y 523.482,Z 275.269,A -85,B 0,C 180,E1 -4753.442,E2 -4753.442} C_VEL
LIN {X 0,Y 526.339,Z 289.551,A -85,B 0,C 180,E1 -4753.829,E2 -4753.829} C_VEL
LIN {X 0,Y 526.097,Z 301.697,A -85,B 0,C 180,E1 -4754.199,E2 -4754.199} C_VEL
LIN {X 0,Y 525.769,Z 313.799,A -85,B 0,C 180,E1 -4754.692,E2 -4754.692} C_VEL
LIN {X 0,Y 525.374,Z 326.713,A -85,B 0,C 180,E1 -4755.375,E2 -4755.375} C_VEL
LIN {X 0,Y 524.972,Z 339.825,A -85,B 0,C 180,E1 -4756.253,E2 -4756.253} C_VEL
LIN {X 0,Y 524.65,Z 351.608,A -85,B 0,C 180,E1 -4757.23,E2 -4757.23} C_VEL
LIN {X 0,Y 524.378,Z 361.505,A -85,B 0,C 180,E1 -4758.221,E2 -4758.221} C_VEL
LIN {X 0,Y 524.058,Z 371.128,A -85,B 0,C 180,E1 -4759.374,E2 -4759.374} C_VEL
LIN {X 0,Y 523.843,Z 379.226,A -85,B 0,C 180,E1 -4760.54,E2 -4760.54} C_VEL
LIN {X 0,Y 523.611,Z 386.988,A -85,B 0,C 180,E1 -4761.898,E2 -4761.898} C_VEL
LIN {X 0,Y 523.53,Z 393.876,A -85,B 0,C 180,E1 -4763.412,E2 -4763.412} C_VEL
LIN {X 0,Y 523.451,Z 398.108,A -85,B 0,C 180,E1 -4764.607,E2 -4764.607} C_VEL
LIN {X 0,Y 523.419,Z 402.244,A -85,B 0,C 180,E1 -4766.15,E2 -4766.15} C_VEL
LIN {X 0,Y 523.333,Z 404.944,A -85,B 0,C 180,E1 -4767.691,E2 -4767.691} C_VEL
LIN {X 0,Y 523.245,Z 406.281,A -85,B 0,C 180,E1 -4769.23,E2 -4769.23} C_VEL
LIN {X 0,Y 523.245,Z 406.281,A -85,B 0,C 180,E1 -4770.77,E2 -4770.77} C_VEL
LIN {X 0,Y 523.333,Z 404.947,A -85,B 0,C 180,E1 -4772.309,E2 -4772.309} C_VEL
LIN {X 0,Y 523.419,Z 402.248,A -85,B 0,C 180,E1 -4773.849,E2 -4773.849} C_VEL
LIN {X 0,Y 523.452,Z 398.109,A -85,B 0,C 180,E1 -4775.393,E2 -4775.393} C_VEL
LIN {X 0,Y 523.495,Z 392.406,A -85,B 0,C 180,E1 -4776.94,E2 -4776.94} C_VEL
LIN {X 0,Y 523.635,Z 385.977,A -85,B 0,C 180,E1 -4778.296,E2 -4778.296} C_VEL
LIN {X 0,Y 523.854,Z 377.991,A -85,B 0,C 180,E1 -4779.654,E2 -4779.654} C_VEL
LIN {X 0,Y 524.106,Z 369.638,A -85,B 0,C 180,E1 -4780.82,E2 -4780.82} C_VEL
LIN {X 0,Y 524.445,Z 358.839,A -85,B 0,C 180,E1 -4782.068,E2 -4782.068} C_VEL
LIN {X 0,Y 524.744,Z 348.366,A -85,B 0,C 180,E1 -4783.062,E2 -4783.062} C_VEL
LIN {X 0,Y 525.101,Z 335.783,A -85,B 0,C 180,E1 -4784.039,E2 -4784.039} C_VEL
LIN {X 0,Y 525.512,Z 323.293,A -85,B 0,C 180,E1 -4784.819,E2 -4784.819} C_VEL
LIN {X 0,Y 525.912,Z 310.457,A -85,B 0,C 180,E1 -4785.452,E2 -4785.452} C_VEL
LIN {X 0,Y 526.164,Z 296.494,A -85,B 0,C 180,E1 -4785.974,E2 -4785.974} C_VEL
LIN {X 0,Y 526.17,Z 288.288,A -85,B 0,C 180,E1 -4786.211,E2 -4786.211} C_VEL
LIN {X 0,Y 523.472,Z 275.11,A -85,B 0,C 180,E1 -4786.577,E2 -4786.577} C_VEL
LIN {X 0,Y 523.602,Z 267.606,A -85,B 0,C 180,E1 -4789.607,E2 -4789.607} C_VEL
LIN {X 0,Y 523.698,Z 261.255,A -85,B 0,C 180,E1 -4792.184,E2 -4792.184} C_VEL
LIN {X 0,Y 523.803,Z 254.464,A -85,B 0,C 180,E1 -4795.002,E2 -4795.002} C_VEL
LIN {X 0,Y 523.998,Z 247.407,A -85,B 0,C 180,E1 -4797.997,E2 -4797.997} C_VEL
LIN {X 0,Y 524.102,Z 240.815,A -85,B 0,C 180,E1 -4800.883,E2 -4800.883} C_VEL
LIN {X 0,Y 524.258,Z 234.39,A -85,B 0,C 180,E1 -4803.783,E2 -4803.783} C_VEL
LIN {X 0,Y 524.362,Z 228.673,A -85,B 0,C 180,E1 -4806.469,E2 -4806.469} C_VEL
LIN {X 0,Y 524.322,Z 223.576,A -85,B 0,C 180,E1 -4808.974,E2 -4808.974} C_VEL
LIN {X 0,Y 523.968,Z 220.844,A -85,B 0,C 180,E1 -4810.455,E2 -4810.455} C_VEL
LIN {X 0,Y 523.904,Z 220.851,A -85,B 0,C 180,E1 -4813.582,E2 -4813.582} C_VEL
LIN {X 0,Y 523.919,Z 220.852,A -85,B 0,C 180,E1 -4816.417,E2 -4816.417} C_VEL
LIN {X 0,Y 523.942,Z 220.845,A -85,B 0,C 180,E1 -4818.908,E2 -4818.908} C_VEL
LIN {X 0,Y 523.914,Z 220.848,A -85,B 0,C 180,E1 -4821.898,E2 -4821.898} C_VEL
LIN {X 0,Y 523.923,Z 220.848,A -85,B 0,C 180,E1 -4824.912,E2 -4824.912} C_VEL
LIN {X 0,Y 523.94,Z 220.849,A -85,B 0,C 180,E1 -4827.679,E2 -4827.679} C_VEL
LIN {X 0,Y 523.953,Z 220.847,A -85,B 0,C 180,E1 -4830.677,E2 -4830.677} C_VEL
LIN {X 0,Y 523.929,Z 220.848,A -85,B 0,C 180,E1 -4833.726,E2 -4833.726} C_VEL
LIN {X 0,Y 523.914,Z 220.848,A -85,B 0,C 180,E1 -4836.27,E2 -4836.27} C_VEL
LIN {X 0,Y 523.948,Z 220.848,A -85,B 0,C 180,E1 -4838.767,E2 -4838.767} C_VEL
LIN {X 0,Y 523.936,Z 220.844,A -85,B 0,C 180,E1 -4841.22,E2 -4841.22} C_VEL
LIN {X 0,Y 523.906,Z 220.852,A -85,B 0,C 180,E1 -4843.638,E2 -4843.638} C_VEL
LIN {X 0,Y 523.947,Z 220.842,A -85,B 0,C 180,E1 -4846.028,E2 -4846.028} C_VEL
LIN {X 0,Y 524.015,Z 220.838,A -85,B 0,C 180,E1 -4848.394,E2 -4848.394} C_VEL
LIN {X 0,Y 523.956,Z 220.844,A -85,B 0,C 180,E1 -4851.515,E2 -4851.515} C_VEL
LIN {X 0,Y 524.07,Z 220.828,A -85,B 0,C 180,E1 -4854.614,E2 -4854.614} C_VEL
LIN {X 0,Y 524.113,Z 220.822,A -85,B 0,C 180,E1 -4857.695,E2 -4857.695} C_VEL
LIN {X 0,Y 524.119,Z 220.822,A -85,B 0,C 180,E1 -4860.768,E2 -4860.768} C_VEL
LIN {X 0,Y 524.039,Z 220.836,A -85,B 0,C 180,E1 -4863.075,E2 -4863.075} C_VEL
LIN {X 0,Y 524.04,Z 220.834,A -85,B 0,C 180,E1 -4866.159,E2 -4866.159} C_VEL
LIN {X 0,Y 524.004,Z 220.837,A -85,B 0,C 180,E1 -4868.484,E2 -4868.484} C_VEL
LIN {X 0,Y 524.001,Z 220.838,A -85,B 0,C 180,E1 -4871.737,E2 -4871.737} C_VEL
LIN {X 0,Y 523.993,Z 220.838,A -85,B 0,C 180,E1 -4875.051,E2 -4875.051} C_VEL
LIN {X 0,Y 523.966,Z 220.845,A -85,B 0,C 180,E1 -4877.969,E2 -4877.969} C_VEL
LIN {X 0,Y 523.96,Z 220.841,A -85,B 0,C 180,E1 -4880.411,E2 -4880.411} C_VEL
LIN {X 0,Y 523.91,Z 220.851,A -85,B 0,C 180,E1 -4882.894,E2 -4882.894} C_VEL
LIN {X 0,Y 523.986,Z 220.843,A -85,B 0,C 180,E1 -4886.02,E2 -4886.02} C_VEL
LIN {X 0,Y 523.931,Z 220.847,A -85,B 0,C 180,E1 -4888.875,E2 -4888.875} C_VEL
LIN {X 0,Y 523.921,Z 220.846,A -85,B 0,C 180,E1 -4891.544,E2 -4891.544} C_VEL
LIN {X 0,Y 523.923,Z 220.849,A -85,B 0,C 180,E1 -4894.291,E2 -4894.291} C_VEL
LIN {X 0,Y 523.909,Z 220.852,A -85,B 0,C 180,E1 -4897.132,E2 -4897.132} C_VEL
LIN {X 0,Y 523.914,Z 220.848,A -85,B 0,C 180,E1 -4900.127,E2 -4900.127} C_VEL
LIN {X 0,Y 523.903,Z 220.85,A -85,B 0,C 180,E1 -4903.169,E2 -4903.169} C_VEL
LIN {X 0,Y 523.933,Z 220.847,A -85,B 0,C 180,E1 -4905.771,E2 -4905.771} C_VEL
LIN {X 0,Y 523.917,Z 220.851,A -85,B 0,C 180,E1 -4906.914,E2 -4906.914} C_VEL
LIN {X 0,Y 523.248,Z 220.933,A -85,B 0,C 180,E1 -4907.555,E2 -4907.555} C_VEL
LIN {X 0,Y 520.392,Z 221.293,A -85,B 0,C 180,E1 -4908.597,E2 -4908.597} C_VEL
LIN {X 0,Y 517.977,Z 221.595,A -85,B 0,C 180,E1 -4909.436,E2 -4909.436} C_VEL
LIN {X 0,Y 516.939,Z 221.723,A -85,B 0,C 180,E1 -4910.084,E2 -4910.084} C_VEL
LIN {X 0,Y 516.854,Z 221.732,A -85,B 0,C 180,E1 -4910.303,E2 -4910.303} C_VEL
LIN {X 0,Y 516.868,Z 221.985,A -85,B 0,C 180,E1 -4911.283,E2 -4911.283} C_VEL
LIN {X 0,Y 516.909,Z 226.318,A -85,B 0,C 180,E1 -4914.223,E2 -4914.223} C_VEL
LIN {X 0,Y 516.782,Z 230.623,A -85,B 0,C 180,E1 -4917.045,E2 -4917.045} C_VEL
LIN {X 0,Y 516.677,Z 234.905,A -85,B 0,C 180,E1 -4919.782,E2 -4919.782} C_VEL
LIN {X 0,Y 516.589,Z 239.165,A -85,B 0,C 180,E1 -4922.448,E2 -4922.448} C_VEL
LIN {X 0,Y 516.555,Z 243.411,A -85,B 0,C 180,E1 -4925.054,E2 -4925.054} C_VEL
LIN {X 0,Y 516.492,Z 247.859,A -85,B 0,C 180,E1 -4927.712,E2 -4927.712} C_VEL
LIN {X 0,Y 516.438,Z 252.009,A -85,B 0,C 180,E1 -4930.11,E2 -4930.11} C_VEL
LIN {X 0,Y 516.426,Z 257.472,A -85,B 0,C 180,E1 -4933.267,E2 -4933.267} C_VEL
LIN {X 0,Y 519.49,Z 271.444,A -85,B 0,C 180,E1 -4933.681,E2 -4933.681} C_VEL
LIN {X 0,Y 519.27,Z 285.107,A -85,B 0,C 180,E1 -4934.128,E2 -4934.128} C_VEL
LIN {X 0,Y 518.906,Z 297.762,A -85,B 0,C 180,E1 -4934.686,E2 -4934.686} C_VEL
LIN {X 0,Y 518.515,Z 310.006,A -85,B 0,C 180,E1 -4935.378,E2 -4935.378} C_VEL
LIN {X 0,Y 518.109,Z 322.603,A -85,B 0,C 180,E1 -4936.268,E2 -4936.268} C_VEL
LIN {X 0,Y 517.693,Z 333.973,A -85,B 0,C 180,E1 -4937.256,E2 -4937.256} C_VEL
LIN {X 0,Y 517.35,Z 343.396,A -85,B 0,C 180,E1 -4938.243,E2 -4938.243} C_VEL
LIN {X 0,Y 517.014,Z 352.859,A -85,B 0,C 180,E1 -4939.426,E2 -4939.426} C_VEL
LIN {X 0,Y 516.735,Z 361.888,A -85,B 0,C 180,E1 -4940.804,E2 -4940.804} C_VEL
LIN {X 0,Y 516.542,Z 369.155,A -85,B 0,C 180,E1 -4942.18,E2 -4942.18} C_VEL
LIN {X 0,Y 516.403,Z 375.682,A -85,B 0,C 180,E1 -4943.75,E2 -4943.75} C_VEL
LIN {X 0,Y 516.306,Z 379.519,A -85,B 0,C 180,E1 -4944.924,E2 -4944.924} C_VEL
LIN {X 0,Y 516.343,Z 382.46,A -85,B 0,C 180,E1 -4946.098,E2 -4946.098} C_VEL
LIN {X 0,Y 516.259,Z 385.171,A -85,B 0,C 180,E1 -4947.659,E2 -4947.659} C_VEL
LIN {X 0,Y 516.156,Z 386.534,A -85,B 0,C 180,E1 -4949.22,E2 -4949.22} C_VEL
LIN {X 0,Y 516.158,Z 386.577,A -85,B 0,C 180,E1 -4950.78,E2 -4950.78} C_VEL
LIN {X 0,Y 516.258,Z 385.295,A -85,B 0,C 180,E1 -4952.341,E2 -4952.341} C_VEL
LIN {X 0,Y 516.343,Z 382.66,A -85,B 0,C 180,E1 -4953.902,E2 -4953.902} C_VEL
LIN {X 0,Y 516.385,Z 378.605,A -85,B 0,C 180,E1 -4955.467,E2 -4955.467} C_VEL
LIN {X 0,Y 516.44,Z 373.003,A -85,B 0,C 180,E1 -4957.035,E2 -4957.035} C_VEL
LIN {X 0,Y 516.606,Z 366.674,A -85,B 0,C 180,E1 -4958.409,E2 -4958.409} C_VEL
LIN {X 0,Y 516.82,Z 358.804,A -85,B 0,C 180,E1 -4959.787,E2 -4959.787} C_VEL
LIN {X 0,Y 517.126,Z 350.57,A -85,B 0,C 180,E1 -4960.968,E2 -4960.968} C_VEL
LIN {X 0,Y 517.485,Z 340.558,A -85,B 0,C 180,E1 -4962.162,E2 -4962.162} C_VEL
LIN {X 0,Y 517.856,Z 329.603,A -85,B 0,C 180,E1 -4963.239,E2 -4963.239} C_VEL
